C07304=1180.329,132.790,-53.848,-178.564,6.325,148.723
C07305=1180.334,132.522,-53.826,-178.567,6.323,148.724
C07306=1180.340,132.253,-53.804,-178.570,6.322,148.724
C07307=1180.345,131.985,-53.783,-178.573,6.320,148.725
C07308=1180.349,131.735,-53.763,-178.576,6.319,148.725
C07309=1180.354,131.487,-53.743,-178.578,6.318,148.726
C07310=1180.360,131.238,-53.722,-178.581,6.316,148.726
C07311=1180.364,130.988,-53.703,-178.583,6.314,148.726
C07312=1180.369,130.739,-53.682,-178.586,6.313,148.727
C07313=1180.374,130.489,-53.663,-178.589,6.311,148.727
C07314=1180.379,130.241,-53.643,-178.591,6.310,148.728
C07315=1180.383,129.992,-53.623,-178.594,6.308,148.728
C07316=1180.388,129.742,-53.603,-178.597,6.307,148.729
C07317=1180.392,129.493,-53.583,-178.600,6.305,148.729
C07318=1180.398,129.244,-53.564,-178.602,6.304,148.730
C07319=1180.402,128.995,-53.543,-178.605,6.302,148.730
C07320=1180.407,128.746,-53.524,-178.607,6.301,148.730
C07321=1180.411,128.497,-53.503,-178.611,6.299,148.731
C07322=1180.416,128.247,-53.484,-178.613,6.298,148.731
C07323=1180.422,127.998,-53.464,-178.615,6.297,148.732
C07324=1180.426,127.749,-53.444,-178.618,6.295,148.732
C07325=1180.431,127.500,-53.424,-178.621,6.294,148.733
C07326=1180.435,127.250,-53.405,-178.623,6.293,148.733
C07327=1180.440,127.002,-53.385,-178.626,6.291,148.734
C07328=1180.445,126.752,-53.365,-178.629,6.289,148.734
C07329=1180.450,126.503,-53.345,-178.631,6.289,148.735
C07330=1180.454,126.254,-53.325,-178.634,6.287,148.735
C07331=1180.460,126.005,-53.306,-178.637,6.285,148.735
C07332=1180.465,125.756,-53.286,-178.640,6.283,148.736
C07333=1180.469,125.507,-53.266,-178.642,6.283,148.736
C07334=1180.474,125.258,-53.246,-178.645,6.281,148.737
C07335=1180.479,125.008,-53.227,-178.648,6.279,148.737
C07336=1180.484,124.759,-53.207,-178.650,6.278,148.738
C07337=1180.488,124.510,-53.187,-178.653,6.277,148.738
C07338=1180.493,124.261,-53.168,-178.656,6.275,148.739
C07339=1180.498,124.012,-53.148,-178.658,6.273,148.739
C07340=1180.502,123.762,-53.129,-178.660,6.273,148.739
C07341=1180.508,123.513,-53.109,-178.664,6.271,148.740
C07342=1180.512,123.264,-53.089,-178.666,6.269,148.740
C07343=1180.517,123.015,-53.069,-178.669,6.268,148.741
C07344=1180.522,122.766,-53.050,-178.671,6.267,148.741
C07345=1180.527,122.516,-53.030,-178.674,6.265,148.742
C07346=1180.531,122.267,-53.011,-178.677,6.264,148.742
C07347=1180.536,122.018,-52.992,-178.679,6.263,148.743
C07348=1180.541,121.768,-52.972,-178.682,6.261,148.743
C07349=1180.545,121.519,-52.952,-178.685,6.260,148.744
C07350=1180.551,121.271,-52.933,-178.687,6.259,148.744
C07351=1180.556,121.021,-52.913,-178.690,6.257,148.745
C07352=1180.560,120.773,-52.894,-178.693,6.256,148.745
C07353=1180.565,120.523,-52.875,-178.695,6.255,148.746
C07354=1180.570,120.273,-52.855,-178.698,6.253,148.746
C07355=1180.575,120.024,-52.836,-178.701,6.251,148.747
C07356=1180.580,119.775,-52.816,-178.704,6.250,148.747
C07357=1180.584,119.526,-52.797,-178.706,6.249,148.747
C07358=1180.589,119.277,-52.778,-178.709,6.247,148.748
C07359=1180.594,119.027,-52.758,-178.712,6.246,148.748
C07360=1180.599,118.778,-52.739,-178.714,6.245,148.749
C07361=1180.603,118.529,-52.720,-178.717,6.243,148.749
C07362=1180.608,118.280,-52.700,-178.720,6.242,148.750
C07363=1180.613,118.031,-52.681,-178.722,6.241,148.750
C07364=1180.617,117.781,-52.662,-178.725,6.239,148.751
C07365=1180.623,117.533,-52.642,-178.727,6.237,148.751
C07366=1180.627,117.283,-52.623,-178.730,6.237,148.752
C07367=1180.633,117.034,-52.604,-178.733,6.235,148.752
C07368=1180.637,116.785,-52.584,-178.735,6.233,148.753
C07369=1180.642,116.536,-52.565,-178.738,6.233,148.753
C07370=1180.647,116.286,-52.546,-178.741,6.231,148.754
C07371=1180.652,116.037,-52.528,-178.743,6.229,148.754
C07372=1180.656,115.788,-52.508,-178.746,6.229,148.755
C07373=1180.661,115.538,-52.488,-178.749,6.227,148.755
C07374=1180.666,115.290,-52.470,-178.751,6.225,148.755
C07375=1180.671,115.040,-52.450,-178.753,6.224,148.756
C07376=1180.676,114.791,-52.431,-178.757,6.223,148.756
C07377=1180.680,114.542,-52.412,-178.759,6.221,148.757
C07378=1180.686,114.292,-52.393,-178.762,6.220,148.757
C07379=1180.690,114.043,-52.373,-178.765,6.219,148.758
C07380=1180.695,113.794,-52.355,-178.767,6.217,148.758
C07381=1180.700,113.545,-52.335,-178.770,6.216,148.759
C07382=1180.704,113.296,-52.316,-178.773,6.215,148.759
C07383=1180.709,113.046,-52.297,-178.775,6.214,148.760
C07384=1180.715,112.797,-52.278,-178.778,6.212,148.760
C07385=1180.719,112.549,-52.259,-178.781,6.211,148.761
C07386=1180.724,112.299,-52.240,-178.783,6.210,148.761
C07387=1180.729,112.050,-52.222,-178.786,6.208,148.762
C07388=1180.734,111.800,-52.202,-178.789,6.207,148.762
C07389=1180.738,111.552,-52.183,-178.791,6.206,148.763
C07390=1180.743,111.301,-52.164,-178.794,6.204,148.763
C07391=1180.748,111.053,-52.146,-178.797,6.203,148.764
C07392=1180.753,110.803,-52.126,-178.799,6.202,148.764
C07393=1180.758,110.554,-52.107,-178.802,6.200,148.764
C07394=1180.762,110.305,-52.088,-178.804,6.199,148.765
C07395=1180.768,110.056,-52.069,-178.807,6.198,148.766
C07396=1180.773,109.807,-52.051,-178.810,6.196,148.766
C07397=1180.777,109.557,-52.031,-178.812,6.195,148.767
C07398=1180.782,109.308,-52.013,-178.815,6.194,148.767
C07399=1180.786,109.059,-51.994,-178.817,6.193,148.767
C07400=1180.792,108.810,-51.975,-178.820,6.191,148.768
C07401=1180.796,108.560,-51.957,-178.823,6.190,148.768
C07402=1180.801,108.311,-51.938,-178.825,6.189,148.769
C07403=1180.806,108.062,-51.920,-178.828,6.187,148.769
C07404=1180.811,107.812,-51.900,-178.831,6.186,148.770
C07405=1180.815,107.564,-51.881,-178.834,6.185,148.771
C07406=1180.820,107.313,-51.862,-178.836,6.183,148.771
C07407=1180.825,107.065,-51.844,-178.839,6.182,148.771
C07408=1180.831,106.796,-51.824,-178.842,6.181,148.772
C07409=1180.835,106.527,-51.804,-178.844,6.179,148.772
C07410=1180.841,106.259,-51.783,-178.848,6.178,148.773
C07411=1180.846,105.991,-51.764,-178.850,6.176,148.773
C07412=1180.851,105.742,-51.744,-178.853,6.176,148.774
C07413=1180.856,105.492,-51.726,-178.856,6.174,148.774
C07414=1180.860,105.244,-51.707,-178.858,6.173,148.775
C07415=1180.865,104.994,-51.688,-178.861,6.172,148.776
C07416=1180.870,104.744,-51.670,-178.864,6.170,148.776
C07417=1180.876,104.496,-51.651,-178.866,6.169,148.777
C07418=1180.880,104.246,-51.633,-178.869,6.168,148.777
C07419=1180.884,103.997,-51.614,-178.871,6.167,148.777
C07420=1180.890,103.748,-51.595,-178.874,6.165,148.778
C07421=1180.895,103.499,-51.577,-178.876,6.164,148.778
C07422=1180.899,103.249,-51.558,-178.879,6.163,148.779
C07423=1180.905,103.000,-51.540,-178.882,6.161,148.779
C07424=1180.909,102.751,-51.521,-178.885,6.160,148.780
C07425=1180.914,102.501,-51.503,-178.888,6.159,148.781
C07426=1180.919,102.252,-51.485,-178.890,6.158,148.781
C07427=1180.924,102.003,-51.466,-178.893,6.156,148.781
C07428=1180.928,101.753,-51.447,-178.895,6.156,148.782
C07429=1180.933,101.504,-51.429,-178.898,6.154,148.782
C07430=1180.939,101.255,-51.411,-178.901,6.153,148.783
C07431=1180.943,101.006,-51.392,-178.903,6.152,148.783
C07432=1180.948,100.756,-51.374,-178.906,6.150,148.784
C07433=1180.953,100.507,-51.356,-178.909,6.150,148.785
C07434=1180.958,100.258,-51.336,-178.911,6.148,148.785
C07435=1180.963,100.009,-51.318,-178.914,6.147,148.786
C07436=1180.967,99.759,-51.300,-178.917,6.146,148.786
C07437=1180.972,99.510,-51.282,-178.919,6.145,148.786
C07438=1180.977,99.261,-51.264,-178.922,6.143,148.787
C07439=1180.982,99.012,-51.245,-178.925,6.142,148.787
C07440=1180.987,98.762,-51.226,-178.927,6.141,148.788
C07441=1180.992,98.513,-51.208,-178.930,6.139,148.789
C07442=1180.996,98.264,-51.190,-178.932,6.138,148.789
C07443=1181.001,98.015,-51.172,-178.935,6.137,148.790
C07444=1181.006,97.765,-51.153,-178.937,6.136,148.790
C07445=1181.011,97.516,-51.135,-178.941,6.135,148.791
C07446=1181.016,97.267,-51.117,-178.943,6.134,148.791
C07447=1181.021,97.018,-51.099,-178.946,6.132,148.791
C07448=1181.026,96.768,-51.081,-178.948,6.132,148.792
C07449=1181.030,96.518,-51.063,-178.951,6.130,148.793
C07450=1181.035,96.269,-51.045,-178.953,6.129,148.793
C07451=1181.041,96.020,-51.026,-178.956,6.128,148.794
C07452=1181.046,95.771,-51.008,-178.959,6.126,148.794
C07453=1181.050,95.521,-50.990,-178.962,6.125,148.795
C07454=1181.055,95.273,-50.971,-178.964,6.124,148.795
C07455=1181.059,95.023,-50.953,-178.967,6.123,148.796
C07456=1181.064,94.774,-50.935,-178.970,6.121,148.796
C07457=1181.069,94.525,-50.917,-178.972,6.120,148.797
C07458=1181.074,94.276,-50.899,-178.975,6.119,148.797
C07459=1181.079,94.026,-50.881,-178.977,6.118,148.798
C07460=1181.084,93.777,-50.863,-178.980,6.117,148.798
C07461=1181.088,93.527,-50.845,-178.982,6.116,148.799
C07462=1181.093,93.278,-50.827,-178.986,6.114,148.799
C07463=1181.098,93.029,-50.809,-178.988,6.114,148.800
C07464=1181.103,92.780,-50.791,-178.990,6.112,148.800
C07465=1181.109,92.530,-50.773,-178.993,6.111,148.801
C07466=1181.114,92.280,-50.755,-178.996,6.110,148.801
C07467=1181.119,92.031,-50.737,-178.998,6.109,148.802
C07468=1181.124,91.782,-50.719,-179.001,6.107,148.802
C07469=1181.128,91.532,-50.701,-179.004,6.107,148.803
C07470=1181.133,91.283,-50.683,-179.006,6.105,148.803
C07471=1181.138,91.034,-50.665,-179.009,6.104,148.804
C07472=1181.142,90.785,-50.647,-179.012,6.103,148.804
C07473=1181.147,90.536,-50.629,-179.014,6.102,148.805
C07474=1181.152,90.287,-50.611,-179.017,6.100,148.805
C07475=1181.157,90.037,-50.594,-179.019,6.100,148.806
C07476=1181.162,89.788,-50.576,-179.022,6.098,148.807
C07477=1181.167,89.539,-50.558,-179.025,6.097,148.807
C07478=1181.172,89.289,-50.540,-179.028,6.096,148.808
C07479=1181.177,89.040,-50.522,-179.030,6.095,148.808
C07480=1181.182,88.791,-50.504,-179.033,6.094,148.809
C07481=1181.187,88.541,-50.487,-179.035,6.093,148.809
C07482=1181.191,88.291,-50.469,-179.038,6.091,148.810
C07483=1181.196,88.042,-50.451,-179.041,6.091,148.810
C07484=1181.201,87.793,-50.433,-179.043,6.089,148.811
C07485=1181.206,87.543,-50.415,-179.046,6.088,148.811
C07486=1181.211,87.294,-50.397,-179.049,6.087,148.812
C07487=1181.215,87.045,-50.380,-179.051,6.086,148.812
C07488=1181.220,86.796,-50.362,-179.054,6.084,148.813
C07489=1181.225,86.546,-50.345,-179.057,6.084,148.813
C07490=1181.230,86.297,-50.327,-179.059,6.083,148.814
C07491=1181.235,86.048,-50.309,-179.062,6.082,148.814
C07492=1181.240,85.798,-50.292,-179.064,6.081,148.815
C07493=1181.245,85.549,-50.274,-179.067,6.079,148.815
C07494=1181.249,85.300,-50.256,-179.069,6.078,148.816
C07495=1181.255,85.050,-50.239,-179.072,6.077,148.816
C07496=1181.260,84.801,-50.221,-179.075,6.076,148.817
C07497=1181.265,84.552,-50.203,-179.078,6.074,148.817
C07498=1181.270,84.302,-50.186,-179.080,6.074,148.818
C07499=1181.274,84.053,-50.168,-179.083,6.072,148.819
C07500=1181.279,83.804,-50.150,-179.086,6.072,148.819
C07501=1181.284,83.554,-50.133,-179.088,6.071,148.820
C07502=1181.289,83.305,-50.115,-179.091,6.069,148.820
C07503=1181.294,83.055,-50.098,-179.093,6.068,148.821
C07504=1181.298,82.806,-50.080,-179.096,6.067,148.821
C07505=1181.304,82.557,-50.063,-179.098,6.066,148.822
C07506=1181.309,82.308,-50.046,-179.102,6.065,148.822
C07507=1181.314,82.059,-50.028,-179.104,6.064,148.823
C07508=1181.318,81.809,-50.011,-179.107,6.063,148.823
C07509=1181.323,81.560,-49.993,-179.109,6.062,148.824
C07510=1181.329,81.310,-49.976,-179.111,6.061,148.824
C07511=1181.333,81.062,-49.958,-179.114,6.059,148.825
C07512=1181.338,80.793,-49.940,-179.118,6.058,148.826
C07513=1181.344,80.524,-49.921,-179.120,6.057,148.826
C07514=1181.349,80.256,-49.902,-179.123,6.056,148.827
C07515=1181.355,79.987,-49.883,-179.126,6.055,148.827
C07516=1181.359,79.739,-49.866,-179.128,6.054,148.828
C07517=1181.364,79.489,-49.848,-179.131,6.053,148.828
C07518=1181.369,79.239,-49.831,-179.134,6.051,148.829
C07519=1181.373,78.990,-49.814,-179.136,6.051,148.830
C07520=1181.379,78.741,-49.797,-179.138,6.050,148.830
C07521=1181.384,78.492,-49.779,-179.142,6.049,148.831
C07522=1181.389,78.242,-49.762,-179.144,6.048,148.831
C07523=1181.394,77.993,-49.745,-179.147,6.046,148.832
C07524=1181.399,77.743,-49.727,-179.149,6.045,148.832
C07525=1181.403,77.494,-49.710,-179.152,6.044,148.833
C07526=1181.408,77.245,-49.692,-179.154,6.043,148.833
C07527=1181.413,76.995,-49.676,-179.157,6.043,148.834
C07528=1181.418,76.746,-49.659,-179.160,6.041,148.834
C07529=1181.423,76.497,-49.641,-179.162,6.040,148.835
C07530=1181.428,76.248,-49.624,-179.165,6.039,148.835
C07531=1181.433,75.998,-49.607,-179.168,6.038,148.836
C07532=1181.438,75.748,-49.590,-179.170,6.037,148.836
C07533=1181.442,75.499,-49.572,-179.173,6.036,148.837
C07534=1181.448,75.250,-49.556,-179.175,6.035,148.838
C07535=1181.453,75.000,-49.539,-179.179,6.034,148.838
C07536=1181.458,74.751,-49.521,-179.181,6.033,148.839
C07537=1181.462,74.502,-49.504,-179.183,6.032,148.839
C07538=1181.467,74.252,-49.487,-179.186,6.031,148.840
C07539=1181.472,74.003,-49.470,-179.189,6.030,148.840
C07540=1181.477,73.754,-49.453,-179.191,6.028,148.841
C07541=1181.482,73.505,-49.436,-179.194,6.028,148.841
C07542=1181.487,73.255,-49.419,-179.196,6.027,148.842
C07543=1181.492,73.005,-49.402,-179.199,6.025,148.843
C07544=1181.497,72.756,-49.385,-179.201,6.025,148.843
C07545=1181.502,72.507,-49.368,-179.204,6.024,148.844
C07546=1181.507,72.258,-49.350,-179.207,6.022,148.844
C07547=1181.511,72.008,-49.334,-179.209,6.022,148.845
C07548=1181.516,71.758,-49.316,-179.212,6.020,148.845
C07549=1181.522,71.509,-49.300,-179.215,6.020,148.846
C07550=1181.527,71.260,-49.283,-179.217,6.019,148.846
C07551=1181.531,71.010,-49.266,-179.220,6.017,148.847
C07552=1181.536,70.761,-49.248,-179.222,6.016,148.847
C07553=1181.541,70.512,-49.232,-179.225,6.016,148.848
C07554=1181.546,70.263,-49.215,-179.228,6.015,148.849
C07555=1181.551,70.013,-49.198,-179.230,6.014,148.849
C07556=1181.555,69.763,-49.181,-179.234,6.012,148.850
C07557=1181.561,69.514,-49.164,-179.236,6.011,148.850
C07558=1181.566,69.265,-49.148,-179.238,6.011,148.851
C07559=1181.571,69.015,-49.130,-179.241,6.009,148.851
C07560=1181.576,68.766,-49.114,-179.244,6.009,148.852
C07561=1181.580,68.517,-49.097,-179.246,6.008,148.852
C07562=1181.586,68.267,-49.080,-179.249,6.006,148.853
C07563=1181.590,68.018,-49.064,-179.251,6.006,148.853
C07564=1181.595,67.769,-49.047,-179.254,6.005,148.854
C07565=1181.600,67.519,-49.030,-179.257,6.003,148.855
C07566=1181.605,67.269,-49.013,-179.259,6.003,148.855
C07567=1181.610,67.021,-48.997,-179.262,6.002,148.856
C07568=1181.615,66.771,-48.980,-179.265,6.001,148.856
C07569=1181.620,66.521,-48.963,-179.267,6.000,148.857
C07570=1181.625,66.273,-48.947,-179.270,5.998,148.857
C07571=1181.630,66.023,-48.930,-179.273,5.998,148.858
C07572=1181.634,65.773,-48.913,-179.275,5.997,148.858
C07573=1181.640,65.525,-48.897,-179.278,5.996,148.859
C07574=1181.645,65.275,-48.879,-179.280,5.995,148.860
C07575=1181.649,65.025,-48.863,-179.283,5.994,148.860
C07576=1181.655,64.776,-48.847,-179.285,5.993,148.861
C07577=1181.660,64.526,-48.830,-179.288,5.992,148.861
C07578=1181.664,64.277,-48.813,-179.291,5.991,148.862
C07579=1181.669,64.028,-48.797,-179.293,5.990,148.862
C07580=1181.674,63.778,-48.780,-179.296,5.989,148.863
C07581=1181.679,63.529,-48.763,-179.298,5.988,148.863
C07582=1181.684,63.280,-48.747,-179.301,5.987,148.864
C07583=1181.689,63.030,-48.731,-179.304,5.986,148.865
C07584=1181.694,62.781,-48.714,-179.306,5.986,148.865
C07585=1181.699,62.531,-48.697,-179.308,5.985,148.866
C07586=1181.704,62.282,-48.680,-179.312,5.983,148.866
C07587=1181.709,62.033,-48.664,-179.314,5.983,148.867
C07588=1181.714,61.783,-48.648,-179.316,5.982,148.867
C07589=1181.719,61.534,-48.632,-179.320,5.981,148.868
C07590=1181.724,61.284,-48.615,-179.322,5.980,148.869
C07591=1181.728,61.035,-48.598,-179.324,5.979,148.869
C07592=1181.734,60.785,-48.582,-179.327,5.978,148.870
C07593=1181.738,60.536,-48.566,-179.330,5.977,148.870
C07594=1181.743,60.287,-48.549,-179.332,5.976,148.871
C07595=1181.749,60.037,-48.532,-179.335,5.975,148.871
C07596=1181.754,59.788,-48.516,-179.338,5.974,148.872
C07597=1181.758,59.538,-48.500,-179.340,5.973,148.872
C07598=1181.763,59.289,-48.483,-179.343,5.972,148.873
C07599=1181.768,59.039,-48.468,-179.345,5.971,148.874
C07600=1181.773,58.790,-48.451,-179.348,5.971,148.874
C07601=1181.779,58.541,-48.434,-179.350,5.970,148.875
C07602=1181.783,58.291,-48.418,-179.353,5.968,148.875
C07603=1181.788,58.042,-48.402,-179.356,5.968,148.876
C07604=1181.793,57.792,-48.385,-179.358,5.967,148.876
C07605=1181.798,57.543,-48.369,-179.361,5.966,148.877
C07606=1181.803,57.294,-48.353,-179.363,5.965,148.878
C07607=1181.808,57.044,-48.337,-179.366,5.964,148.878
C07608=1181.813,56.795,-48.321,-179.369,5.964,148.879
C07609=1181.818,56.546,-48.304,-179.371,5.962,148.879
C07610=1181.823,56.296,-48.288,-179.374,5.962,148.880
C07611=1181.828,56.047,-48.271,-179.376,5.961,148.880
C07612=1181.833,55.797,-48.255,-179.379,5.959,148.881
C07613=1181.838,55.548,-48.239,-179.381,5.958,148.882
C07614=1181.843,55.298,-48.223,-179.384,5.958,148.882
C07615=1181.848,55.049,-48.207,-179.387,5.957,148.883
C07616=1181.853,54.780,-48.189,-179.389,5.956,148.883
C07617=1181.859,54.511,-48.172,-179.392,5.955,148.884
C07618=1181.864,54.243,-48.155,-179.395,5.954,148.885
C07619=1181.869,53.975,-48.138,-179.398,5.953,148.885
C07620=1181.874,53.725,-48.122,-179.400,5.952,148.886
C07621=1181.879,53.476,-48.105,-179.403,5.951,148.886
C07622=1181.884,53.226,-48.089,-179.406,5.951,148.887
C07623=1181.889,52.977,-48.073,-179.408,5.950,148.888
C07624=1181.894,52.727,-48.057,-179.411,5.949,148.888
C07625=1181.899,52.478,-48.041,-179.414,5.948,148.889
C07626=1181.904,52.228,-48.025,-179.416,5.947,148.889
C07627=1181.909,51.979,-48.009,-179.419,5.947,148.890
C07628=1181.914,51.730,-47.993,-179.422,5.945,148.890
C07629=1181.919,51.480,-47.977,-179.424,5.944,148.891
C07630=1181.924,51.231,-47.961,-179.426,5.943,148.892
C07631=1181.929,50.981,-47.945,-179.429,5.943,148.892
C07632=1181.934,50.732,-47.929,-179.432,5.941,148.893
C07633=1181.939,50.482,-47.913,-179.434,5.941,148.893
C07634=1181.944,50.233,-47.897,-179.437,5.940,148.894
C07635=1181.949,49.984,-47.881,-179.439,5.939,148.894
C07636=1181.953,49.734,-47.865,-179.442,5.938,148.895
C07637=1181.959,49.485,-47.850,-179.445,5.938,148.896
C07638=1181.963,49.235,-47.833,-179.447,5.937,148.896
C07639=1181.969,48.986,-47.818,-179.450,5.936,148.897
C07640=1181.974,48.736,-47.802,-179.452,5.935,148.897
C07641=1181.978,48.487,-47.785,-179.455,5.934,148.898
C07642=1181.984,48.238,-47.770,-179.458,5.933,148.899
C07643=1181.989,47.988,-47.754,-179.460,5.933,148.899
C07644=1181.993,47.738,-47.739,-179.463,5.932,148.900
C07645=1181.998,47.490,-47.722,-179.465,5.930,148.900
C07646=1182.003,47.239,-47.706,-179.468,5.930,148.901
C07647=1182.009,46.990,-47.691,-179.471,5.929,148.902
C07648=1182.014,46.741,-47.675,-179.473,5.928,148.902
C07649=1182.018,46.491,-47.659,-179.476,5.927,148.903
C07650=1182.023,46.242,-47.644,-179.478,5.926,148.903
C07651=1182.028,45.993,-47.628,-179.481,5.926,148.904
C07652=1182.033,45.743,-47.612,-179.483,5.925,148.904
C07653=1182.039,45.493,-47.597,-179.486,5.924,148.905
C07654=1182.044,45.244,-47.580,-179.489,5.923,148.906
C07655=1182.048,44.995,-47.565,-179.491,5.922,148.906
C07656=1182.053,44.745,-47.549,-179.494,5.922,148.907
C07657=1182.059,44.496,-47.534,-179.496,5.921,148.907
C07658=1182.064,44.246,-47.518,-179.499,5.919,148.908
C07659=1182.068,43.997,-47.503,-179.502,5.919,148.908
C07660=1182.073,43.747,-47.487,-179.504,5.918,148.909
C07661=1182.079,43.498,-47.472,-179.506,5.918,148.910
C07662=1182.083,43.248,-47.455,-179.509,5.917,148.910
C07663=1182.088,42.999,-47.440,-179.512,5.915,148.911
C07664=1182.093,42.750,-47.424,-179.514,5.915,148.911
C07665=1182.099,42.500,-47.409,-179.517,5.914,148.912
C07666=1182.103,42.250,-47.393,-179.519,5.913,148.912
C07667=1182.108,42.001,-47.378,-179.522,5.913,148.913
C07668=1182.113,41.752,-47.362,-179.525,5.912,148.914
C07669=1182.118,41.502,-47.346,-179.527,5.911,148.914
C07670=1182.123,41.253,-47.331,-179.530,5.910,148.915
C07671=1182.128,41.003,-47.316,-179.532,5.909,148.915
C07672=1182.134,40.754,-47.300,-179.535,5.909,148.916
C07673=1182.138,40.504,-47.284,-179.538,5.908,148.917
C07674=1182.143,40.255,-47.269,-179.540,5.907,148.917
C07675=1182.148,40.005,-47.254,-179.543,5.906,148.918
C07676=1182.154,39.756,-47.238,-179.545,5.906,148.918
C07677=1182.159,39.507,-47.223,-179.547,5.905,148.919
C07678=1182.163,39.257,-47.207,-179.550,5.904,148.920
C07679=1182.169,39.007,-47.191,-179.553,5.903,148.920
C07680=1182.173,38.758,-47.176,-179.556,5.902,148.921
C07681=1182.179,38.509,-47.161,-179.558,5.902,148.921
C07682=1182.183,38.259,-47.145,-179.560,5.901,148.922
C07683=1182.188,38.010,-47.130,-179.563,5.900,148.923
C07684=1182.194,37.760,-47.114,-179.566,5.900,148.923
C07685=1182.198,37.511,-47.099,-179.568,5.898,148.924
C07686=1182.204,37.261,-47.084,-179.571,5.898,148.924
C07687=1182.209,37.012,-47.069,-179.574,5.897,148.925
C07688=1182.213,36.762,-47.053,-179.576,5.896,148.925
C07689=1182.219,36.512,-47.038,-179.578,5.896,148.926
C07690=1182.223,36.263,-47.023,-179.582,5.894,148.927
C07691=1182.229,36.014,-47.007,-179.584,5.893,148.927
C07692=1182.233,35.765,-46.992,-179.586,5.893,148.928
C07693=1182.239,35.515,-46.977,-179.589,5.892,148.928
C07694=1182.243,35.265,-46.962,-179.591,5.892,148.929
C07695=1182.249,35.016,-46.946,-179.594,5.891,148.930
C07696=1182.254,34.766,-46.931,-179.596,5.890,148.930
C07697=1182.259,34.517,-46.916,-179.599,5.889,148.931
C07698=1182.264,34.267,-46.901,-179.602,5.888,148.931
C07699=1182.269,34.018,-46.886,-179.604,5.888,148.932
C07700=1182.274,33.768,-46.870,-179.607,5.887,148.933
C07701=1182.278,33.519,-46.855,-179.609,5.887,148.933
C07702=1182.284,33.269,-46.840,-179.612,5.886,148.934
C07703=1182.289,33.020,-46.825,-179.615,5.884,148.934
C07704=1182.294,32.770,-46.810,-179.617,5.884,148.935
C07705=1182.299,32.521,-46.795,-179.620,5.883,148.936
C07706=1182.304,32.271,-46.780,-179.622,5.883,148.936
C07707=1182.309,32.022,-46.765,-179.625,5.882,148.937
C07708=1182.314,31.773,-46.749,-179.627,5.881,148.937
C07709=1182.319,31.522,-46.735,-179.630,5.881,148.938
C07710=1182.323,31.273,-46.720,-179.633,5.879,148.939
C07711=1182.329,31.024,-46.704,-179.635,5.878,148.939
C07712=1182.334,30.774,-46.690,-179.638,5.878,148.940
C07713=1182.339,30.525,-46.674,-179.640,5.877,148.940
C07714=1182.344,30.276,-46.659,-179.642,5.877,148.941
C07715=1182.350,30.026,-46.644,-179.645,5.876,148.942
C07716=1182.354,29.776,-46.629,-179.647,5.875,148.942
C07717=1182.359,29.527,-46.614,-179.650,5.875,148.943
C07718=1182.365,29.277,-46.599,-179.653,5.873,148.943
C07719=1182.369,29.028,-46.584,-179.655,5.873,148.944
C07720=1182.375,28.759,-46.568,-179.658,5.872,148.945
C07721=1182.380,28.490,-46.552,-179.661,5.872,148.945
C07722=1182.386,28.221,-46.536,-179.664,5.870,148.946
C07723=1182.391,27.953,-46.520,-179.666,5.870,148.947
C07724=1182.396,27.703,-46.505,-179.669,5.869,148.947
C07725=1182.401,27.454,-46.490,-179.671,5.868,148.948
C07726=1182.406,27.204,-46.476,-179.674,5.868,148.948
C07727=1182.411,26.955,-46.461,-179.677,5.867,148.949
C07728=1182.416,26.705,-46.446,-179.679,5.867,148.950
C07729=1182.421,26.456,-46.431,-179.682,5.865,148.950
C07730=1182.426,26.206,-46.416,-179.685,5.865,148.951
C07731=1182.431,25.957,-46.401,-179.687,5.864,148.951
C07732=1182.436,25.707,-46.387,-179.689,5.863,148.952
C07733=1182.441,25.458,-46.372,-179.692,5.863,148.953
C07734=1182.447,25.208,-46.357,-179.694,5.862,148.953
C07735=1182.451,24.959,-46.342,-179.697,5.862,148.954
C07736=1182.456,24.709,-46.327,-179.700,5.861,148.955
C07737=1182.462,24.460,-46.312,-179.702,5.860,148.955
C07738=1182.467,24.210,-46.298,-179.704,5.860,148.956
C07739=1182.472,23.961,-46.283,-179.708,5.858,148.956
C07740=1182.476,23.711,-46.268,-179.710,5.858,148.957
C07741=1182.482,23.461,-46.253,-179.712,5.857,148.957
C07742=1182.487,23.212,-46.238,-179.715,5.857,148.958
C07743=1182.492,22.963,-46.224,-179.717,5.856,148.959
C07744=1182.497,22.713,-46.210,-179.720,5.855,148.959
C07745=1182.502,22.464,-46.194,-179.722,5.855,148.960
C07746=1182.507,22.214,-46.180,-179.725,5.854,148.960
C07747=1182.512,21.965,-46.165,-179.727,5.853,148.961
C07748=1182.516,21.715,-46.151,-179.730,5.853,148.962
C07749=1182.521,21.465,-46.136,-179.732,5.852,148.962
C07750=1182.527,21.216,-46.121,-179.735,5.851,148.963
C07751=1182.532,20.966,-46.107,-179.738,5.850,148.964
C07752=1182.537,20.716,-46.092,-179.740,5.849,148.964
C07753=1182.541,20.467,-46.077,-179.743,5.849,148.965
C07754=1182.546,20.218,-46.063,-179.745,5.848,148.965
C07755=1182.553,19.968,-46.049,-179.748,5.848,148.966
C07756=1182.558,19.719,-46.034,-179.750,5.847,148.967
C07757=1182.562,19.470,-46.019,-179.753,5.847,148.967
C07758=1182.567,19.220,-46.005,-179.755,5.846,148.968
C07759=1182.572,18.970,-45.991,-179.758,5.845,148.968
C07760=1182.577,18.720,-45.976,-179.760,5.845,148.969
C07761=1182.582,18.471,-45.961,-179.763,5.844,148.969
C07762=1182.587,18.221,-45.947,-179.765,5.843,148.970
C07763=1182.592,17.972,-45.932,-179.768,5.843,148.971
C07764=1182.598,17.723,-45.918,-179.771,5.842,148.972
C07765=1182.603,17.473,-45.903,-179.773,5.841,148.972
C07766=1182.608,17.224,-45.889,-179.776,5.840,148.973
C07767=1182.613,16.974,-45.875,-179.779,5.840,148.973
C07768=1182.617,16.724,-45.861,-179.781,5.839,148.974
C07769=1182.622,16.475,-45.846,-179.783,5.838,148.974
C07770=1182.628,16.225,-45.831,-179.786,5.838,148.975
C07771=1182.633,15.976,-45.816,-179.788,5.837,148.976
C07772=1182.638,15.727,-45.802,-179.791,5.837,148.976
C07773=1182.643,15.477,-45.788,-179.793,5.836,148.977
C07774=1182.648,15.227,-45.774,-179.796,5.835,148.977
C07775=1182.653,14.977,-45.760,-179.798,5.835,148.978
C07776=1182.658,14.728,-45.745,-179.801,5.834,148.979
C07777=1182.663,14.478,-45.731,-179.803,5.833,148.979
C07778=1182.669,14.229,-45.717,-179.806,5.833,148.980
C07779=1182.673,13.980,-45.702,-179.808,5.832,148.981
C07780=1182.678,13.730,-45.688,-179.811,5.832,148.981
C07781=1182.683,13.480,-45.674,-179.813,5.831,148.982
C07782=1182.688,13.231,-45.659,-179.816,5.831,148.982
C07783=1182.694,12.982,-45.645,-179.818,5.830,148.983
C07784=1182.699,12.732,-45.631,-179.821,5.829,148.984
C07785=1182.704,12.482,-45.617,-179.824,5.828,148.984
C07786=1182.709,12.233,-45.603,-179.827,5.828,148.985
C07787=1182.714,11.983,-45.588,-179.829,5.827,148.985
C07788=1182.719,11.734,-45.574,-179.831,5.826,148.986
C07789=1182.724,11.484,-45.560,-179.834,5.826,148.987
C07790=1182.729,11.234,-45.546,-179.836,5.825,148.987
C07791=1182.734,10.985,-45.532,-179.839,5.824,148.988
C07792=1182.740,10.736,-45.518,-179.841,5.824,148.989
C07793=1182.744,10.486,-45.503,-179.844,5.823,148.989
C07794=1182.749,10.236,-45.489,-179.846,5.823,148.990
C07795=1182.754,9.987,-45.475,-179.849,5.822,148.990
C07796=1182.760,9.738,-45.461,-179.852,5.822,148.991
C07797=1182.765,9.488,-45.447,-179.854,5.821,148.992
C07798=1182.770,9.238,-45.432,-179.856,5.820,148.992
C07799=1182.775,8.988,-45.418,-179.859,5.820,148.993
C07800=1182.780,8.739,-45.405,-179.861,5.819,148.993
C07801=1182.785,8.489,-45.391,-179.864,5.818,148.994
C07802=1182.790,8.240,-45.377,-179.867,5.818,148.995
C07803=1182.795,7.990,-45.363,-179.869,5.817,148.995
C07804=1182.800,7.741,-45.349,-179.871,5.817,148.996
C07805=1182.805,7.491,-45.334,-179.874,5.816,148.997
C07806=1182.810,7.242,-45.320,-179.877,5.816,148.997
C07807=1182.815,6.992,-45.306,-179.879,5.815,148.998
C07808=1182.820,6.743,-45.293,-179.881,5.814,148.998
C07809=1182.825,6.493,-45.279,-179.884,5.814,148.999
C07810=1182.830,6.243,-45.265,-179.886,5.813,149.000
C07811=1182.836,5.994,-45.251,-179.889,5.813,149.000
C07812=1182.841,5.744,-45.237,-179.892,5.812,149.001
C07813=1182.846,5.495,-45.222,-179.894,5.811,149.001
C07814=1182.852,5.245,-45.209,-179.896,5.811,149.002
C07815=1182.856,4.996,-45.195,-179.899,5.810,149.003
C07816=1182.861,4.746,-45.181,-179.902,5.810,149.003
C07817=1182.866,4.497,-45.167,-179.904,5.809,149.004
C07818=1182.872,4.247,-45.154,-179.907,5.808,149.005
C07819=1182.877,3.997,-45.139,-179.909,5.808,149.005
C07820=1182.881,3.748,-45.126,-179.911,5.807,149.006
C07821=1182.886,3.499,-45.112,-179.914,5.807,149.006
C07822=1182.892,3.248,-45.098,-179.917,5.806,149.007
C07823=1182.897,2.999,-45.084,-179.919,5.805,149.008
C07824=1182.903,2.730,-45.069,-179.921,5.805,149.008
C07825=1182.907,2.461,-45.055,-179.924,5.804,149.009
C07826=1182.913,2.191,-45.040,-179.927,5.804,149.010
C07827=1182.919,1.923,-45.025,-179.929,5.803,149.010
C07828=1182.924,1.673,-45.011,-179.932,5.803,149.011
C07829=1182.929,1.423,-44.997,-179.935,5.803,149.012
C07830=1182.934,1.173,-44.984,-179.937,5.802,149.012
C07831=1182.939,0.924,-44.970,-179.940,5.801,149.013
C07832=1182.944,0.674,-44.956,-179.942,5.801,149.014
C07833=1182.950,0.425,-44.942,-179.944,5.800,149.014
C07834=1182.954,0.175,-44.929,-179.947,5.799,149.015
C07835=1182.960,-0.074,-44.916,-179.950,5.799,149.015
C07836=1182.965,-0.324,-44.901,-179.952,5.798,149.016
C07837=1182.969,-0.573,-44.888,-179.955,5.798,149.017
C07838=1182.975,-0.823,-44.874,-179.957,5.797,149.017
C07839=1182.980,-1.073,-44.860,-179.960,5.797,149.018
C07840=1182.985,-1.322,-44.847,-179.962,5.796,149.018
C07841=1182.990,-1.572,-44.833,-179.965,5.795,149.019
C07842=1182.995,-1.821,-44.819,-179.967,5.795,149.020
C07843=1183.000,-2.071,-44.806,-179.969,5.794,149.020
C07844=1183.005,-2.321,-44.792,-179.972,5.794,149.021
C07845=1183.011,-2.570,-44.779,-179.975,5.793,149.022
C07846=1183.015,-2.820,-44.765,-179.977,5.793,149.022
C07847=1183.021,-3.069,-44.752,-179.980,5.792,149.023
C07848=1183.026,-3.319,-44.738,-179.982,5.791,149.023
C07849=1183.031,-3.568,-44.725,-179.985,5.791,149.024
C07850=1183.036,-3.818,-44.711,-179.987,5.790,149.025
C07851=1183.042,-4.068,-44.698,-179.990,5.790,149.025
C07852=1183.046,-4.317,-44.684,-179.992,5.789,149.026
C07853=1183.052,-4.567,-44.671,-179.994,5.789,149.027
C07854=1183.056,-4.816,-44.657,-179.997,5.789,149.027
C07855=1183.061,-5.066,-44.644,-179.999,5.788,149.028
C07856=1183.067,-5.315,-44.630,179.998,5.788,149.029
C07857=1183.071,-5.565,-44.617,179.996,5.787,149.029
C07858=1183.077,-5.815,-44.603,179.993,5.786,149.030
C07859=1183.081,-6.064,-44.590,179.991,5.786,149.030
C07860=1183.087,-6.314,-44.577,179.988,5.785,149.031
C07861=1183.091,-6.563,-44.563,179.986,5.785,149.032
C07862=1183.097,-6.813,-44.550,179.983,5.784,149.032
C07863=1183.101,-7.062,-44.536,179.980,5.784,149.033
C07864=1183.107,-7.312,-44.523,179.978,5.783,149.033
C07865=1183.113,-7.562,-44.509,179.976,5.782,149.034
C07866=1183.117,-7.811,-44.496,179.973,5.782,149.035
C07867=1183.123,-8.061,-44.482,179.970,5.781,149.035
C07868=1183.128,-8.311,-44.470,179.968,5.781,149.036
C07869=1183.133,-8.560,-44.456,179.966,5.781,149.037
C07870=1183.138,-8.810,-44.443,179.963,5.780,149.037
C07871=1183.144,-9.059,-44.430,179.961,5.780,149.038
C07872=1183.148,-9.309,-44.416,179.959,5.779,149.038
C07873=1183.154,-9.558,-44.403,179.956,5.779,149.039
C07874=1183.158,-9.808,-44.390,179.953,5.778,149.040
C07875=1183.163,-10.057,-44.377,179.951,5.777,149.040
C07876=1183.168,-10.307,-44.363,179.948,5.777,149.041
C07877=1183.173,-10.557,-44.350,179.946,5.776,149.042
C07878=1183.179,-10.807,-44.337,179.944,5.776,149.042
C07879=1183.184,-11.056,-44.324,179.941,5.775,149.043
C07880=1183.189,-11.305,-44.310,179.938,5.775,149.044
C07881=1183.194,-11.555,-44.297,179.936,5.775,149.044
C07882=1183.200,-11.805,-44.284,179.934,5.774,149.045
C07883=1183.204,-12.054,-44.270,179.931,5.774,149.045
C07884=1183.209,-12.304,-44.258,179.929,5.773,149.046
C07885=1183.214,-12.554,-44.244,179.927,5.772,149.047
C07886=1183.220,-12.803,-44.232,179.924,5.772,149.047
C07887=1183.225,-13.052,-44.218,179.921,5.771,149.048
C07888=1183.230,-13.302,-44.205,179.919,5.771,149.049
C07889=1183.235,-13.552,-44.192,179.916,5.770,149.049
C07890=1183.240,-13.802,-44.179,179.914,5.770,149.050
C07891=1183.245,-14.051,-44.166,179.911,5.769,149.050
C07892=1183.251,-14.301,-44.153,179.909,5.770,149.051
C07893=1183.255,-14.550,-44.139,179.907,5.769,149.052
C07894=1183.260,-14.800,-44.127,179.904,5.768,149.052
C07895=1183.266,-15.049,-44.113,179.902,5.768,149.053
C07896=1183.271,-15.299,-44.100,179.899,5.767,149.053
C07897=1183.276,-15.549,-44.088,179.897,5.767,149.054
C07898=1183.281,-15.799,-44.074,179.894,5.766,149.055
C07899=1183.286,-16.048,-44.062,179.891,5.766,149.056
C07900=1183.291,-16.298,-44.049,179.889,5.765,149.056
C07901=1183.296,-16.547,-44.035,179.887,5.765,149.057
C07902=1183.301,-16.797,-44.022,179.884,5.765,149.057
C07903=1183.307,-17.046,-44.010,179.882,5.764,149.058
C07904=1183.312,-17.296,-43.996,179.880,5.763,149.059
C07905=1183.317,-17.546,-43.983,179.877,5.763,149.059
C07906=1183.322,-17.795,-43.971,179.874,5.762,149.060
C07907=1183.327,-18.045,-43.957,179.872,5.762,149.060
C07908=1183.332,-18.295,-43.945,179.869,5.761,149.061
C07909=1183.338,-18.544,-43.932,179.867,5.761,149.062
C07910=1183.342,-18.794,-43.919,179.865,5.761,149.062
C07911=1183.348,-19.044,-43.906,179.863,5.760,149.063
C07912=1183.353,-19.293,-43.893,179.860,5.760,149.064
C07913=1183.358,-19.542,-43.881,179.857,5.759,149.064
C07914=1183.363,-19.793,-43.867,179.855,5.758,149.065
C07915=1183.369,-20.042,-43.855,179.852,5.758,149.066
C07916=1183.374,-20.291,-43.842,179.850,5.758,149.066
C07917=1183.378,-20.541,-43.829,179.848,5.757,149.067
C07918=1183.384,-20.791,-43.816,179.846,5.757,149.067
C07919=1183.389,-21.040,-43.803,179.843,5.757,149.068
C07920=1183.394,-21.289,-43.791,179.840,5.756,149.069
C07921=1183.399,-21.540,-43.778,179.838,5.755,149.069
C07922=1183.404,-21.789,-43.765,179.835,5.755,149.070
C07923=1183.410,-22.039,-43.753,179.833,5.754,149.071
C07924=1183.415,-22.289,-43.740,179.831,5.754,149.071
C07925=1183.420,-22.538,-43.727,179.828,5.754,149.072
C07926=1183.425,-22.788,-43.714,179.826,5.753,149.072
C07927=1183.430,-23.037,-43.702,179.823,5.753,149.073
C07928=1183.436,-23.307,-43.687,179.820,5.753,149.074
C07929=1183.441,-23.577,-43.674,179.818,5.752,149.075
C07930=1183.447,-23.846,-43.660,179.816,5.751,149.075
C07931=1183.452,-24.117,-43.647,179.813,5.751,149.076
C07932=1183.458,-24.366,-43.634,179.810,5.750,149.076
C07933=1183.463,-24.615,-43.622,179.808,5.750,149.077
C07934=1183.468,-24.865,-43.608,179.805,5.749,149.078
C07935=1183.473,-25.115,-43.596,179.803,5.749,149.078
C07936=1183.478,-25.364,-43.583,179.801,5.749,149.079
C07937=1183.484,-25.614,-43.571,179.798,5.749,149.080
C07938=1183.488,-25.864,-43.558,179.796,5.748,149.080
C07939=1183.493,-26.113,-43.545,179.793,5.747,149.081
C07940=1183.498,-26.363,-43.533,179.791,5.747,149.082
C07941=1183.503,-26.612,-43.520,179.788,5.746,149.082
C07942=1183.509,-26.862,-43.508,179.786,5.746,149.083
C07943=1183.513,-27.112,-43.495,179.784,5.746,149.083
C07944=1183.519,-27.362,-43.482,179.781,5.745,149.084
C07945=1183.524,-27.611,-43.470,179.779,5.745,149.085
C07946=1183.530,-27.861,-43.458,179.776,5.744,149.085
C07947=1183.535,-28.110,-43.445,179.774,5.744,149.086
C07948=1183.540,-28.359,-43.433,179.771,5.744,149.087
C07949=1183.545,-28.610,-43.420,179.769,5.743,149.087
C07950=1183.550,-28.859,-43.408,179.767,5.743,149.088
C07951=1183.555,-29.109,-43.395,179.764,5.742,149.089
C07952=1183.560,-29.358,-43.383,179.762,5.741,149.089
C07953=1183.566,-29.608,-43.371,179.759,5.741,149.090
C07954=1183.571,-29.857,-43.358,179.757,5.741,149.090
C07955=1183.575,-30.107,-43.345,179.754,5.741,149.091
C07956=1183.581,-30.357,-43.333,179.752,5.740,149.092
C07957=1183.586,-30.607,-43.321,179.750,5.740,149.092
C07958=1183.591,-30.856,-43.308,179.747,5.739,149.093
C07959=1183.596,-31.106,-43.296,179.745,5.740,149.094
C07960=1183.602,-31.355,-43.283,179.743,5.739,149.094
C07961=1183.607,-31.605,-43.272,179.740,5.738,149.095
C07962=1183.612,-31.855,-43.259,179.737,5.738,149.096
C07963=1183.617,-32.104,-43.246,179.735,5.737,149.096
C07964=1183.622,-32.354,-43.234,179.732,5.737,149.097
C07965=1183.627,-32.604,-43.222,179.730,5.737,149.097
C07966=1183.633,-32.854,-43.210,179.728,5.736,149.098
C07967=1183.638,-33.103,-43.197,179.726,5.736,149.099
C07968=1183.643,-33.352,-43.184,179.723,5.735,149.099
C07969=1183.648,-33.602,-43.173,179.720,5.735,149.100
C07970=1183.653,-33.852,-43.160,179.719,5.735,149.100
C07971=1183.659,-34.101,-43.148,179.716,5.734,149.101
C07972=1183.663,-34.351,-43.135,179.713,5.734,149.102
C07973=1183.669,-34.601,-43.123,179.711,5.733,149.103
C07974=1183.674,-34.851,-43.111,179.708,5.733,149.103
C07975=1183.679,-35.100,-43.099,179.706,5.733,149.104
C07976=1183.684,-35.350,-43.087,179.704,5.732,149.104
C07977=1183.689,-35.600,-43.075,179.702,5.732,149.105
C07978=1183.694,-35.849,-43.062,179.699,5.731,149.106
C07979=1183.700,-36.099,-43.050,179.696,5.731,149.106
C07980=1183.705,-36.348,-43.038,179.694,5.731,149.107
C07981=1183.710,-36.598,-43.026,179.692,5.730,149.107
C07982=1183.715,-36.847,-43.013,179.689,5.730,149.108
C07983=1183.721,-37.097,-43.001,179.687,5.729,149.109
C07984=1183.726,-37.347,-42.990,179.684,5.729,149.109
C07985=1183.731,-37.596,-42.978,179.682,5.729,149.110
C07986=1183.736,-37.846,-42.966,179.680,5.729,149.111
C07987=1183.741,-38.096,-42.953,179.677,5.728,149.111
C07988=1183.747,-38.346,-42.941,179.675,5.727,149.112
C07989=1183.752,-38.595,-42.929,179.672,5.727,149.113
C07990=1183.757,-38.845,-42.917,179.670,5.727,149.113
C07991=1183.763,-39.095,-42.905,179.668,5.726,149.114
C07992=1183.767,-39.344,-42.893,179.665,5.726,149.114
C07993=1183.772,-39.594,-42.881,179.663,5.725,149.115
C07994=1183.778,-39.844,-42.869,179.661,5.726,149.116
C07995=1183.783,-40.093,-42.856,179.658,5.725,149.116
C07996=1183.788,-40.343,-42.845,179.656,5.725,149.117
C07997=1183.793,-40.592,-42.833,179.653,5.724,149.118
C07998=1183.798,-40.842,-42.821,179.651,5.723,149.118
C07999=1183.804,-41.092,-42.809,179.649,5.724,149.119
C08000=1183.809,-41.341,-42.796,179.646,5.723,149.120
C08001=1183.814,-41.591,-42.784,179.644,5.722,149.120
C08002=1183.819,-41.841,-42.773,179.641,5.722,149.121
C08003=1183.824,-42.091,-42.761,179.639,5.722,149.121
C08004=1183.830,-42.340,-42.748,179.637,5.722,149.122
C08005=1183.835,-42.590,-42.737,179.634,5.721,149.123
C08006=1183.840,-42.839,-42.725,179.632,5.721,149.123
C08007=1183.845,-43.089,-42.713,179.630,5.721,149.124
C08008=1183.850,-43.339,-42.701,179.627,5.720,149.125
C08009=1183.856,-43.589,-42.689,179.625,5.720,149.125
C08010=1183.860,-43.838,-42.678,179.622,5.719,149.126
C08011=1183.865,-44.088,-42.665,179.619,5.719,149.127
C08012=1183.871,-44.337,-42.653,179.618,5.719,149.127
C08013=1183.876,-44.587,-42.642,179.615,5.718,149.128
C08014=1183.881,-44.837,-42.630,179.613,5.718,149.129
C08015=1183.886,-45.087,-42.618,179.610,5.717,149.129
C08016=1183.891,-45.336,-42.606,179.608,5.718,149.130
C08017=1183.896,-45.586,-42.594,179.606,5.717,149.130
C08018=1183.902,-45.836,-42.582,179.603,5.717,149.131
C08019=1183.908,-46.085,-42.571,179.601,5.716,149.132
C08020=1183.912,-46.335,-42.560,179.599,5.716,149.132
C08021=1183.917,-46.584,-42.547,179.596,5.716,149.133
C08022=1183.923,-46.834,-42.535,179.594,5.715,149.133
C08023=1183.928,-47.084,-42.524,179.591,5.715,149.134
C08024=1183.933,-47.334,-42.512,179.589,5.715,149.135
C08025=1183.938,-47.583,-42.500,179.587,5.714,149.135
C08026=1183.943,-47.833,-42.489,179.584,5.714,149.136
C08027=1183.949,-48.083,-42.477,179.582,5.713,149.137
C08028=1183.953,-48.333,-42.465,179.579,5.714,149.137
C08029=1183.959,-48.581,-42.453,179.577,5.713,149.138
C08030=1183.964,-48.831,-42.441,179.575,5.712,149.139
C08031=1183.969,-49.081,-42.430,179.572,5.712,149.139
C08032=1183.975,-49.352,-42.418,179.570,5.712,149.140
C08033=1183.981,-49.621,-42.405,179.568,5.711,149.140
C08034=1183.986,-49.892,-42.392,179.565,5.711,149.141
C08035=1183.991,-50.162,-42.379,179.562,5.711,149.142
C08036=1183.997,-50.412,-42.367,179.560,5.710,149.143
C08037=1184.002,-50.661,-42.356,179.557,5.710,149.143
C08038=1184.007,-50.911,-42.345,179.555,5.710,149.144
C08039=1184.013,-51.161,-42.333,179.553,5.709,149.144
C08040=1184.018,-51.411,-42.321,179.550,5.709,149.145
C08041=1184.023,-51.660,-42.310,179.548,5.709,149.146
C08042=1184.028,-51.910,-42.298,179.546,5.708,149.146
C08043=1184.034,-52.159,-42.287,179.543,5.708,149.147
C08044=1184.038,-52.409,-42.275,179.541,5.708,149.148
C08045=1184.044,-52.659,-42.264,179.539,5.707,149.148
C08046=1184.049,-52.909,-42.252,179.536,5.707,149.149
C08047=1184.054,-53.158,-42.240,179.534,5.707,149.150
C08048=1184.059,-53.408,-42.229,179.531,5.706,149.150
C08049=1184.065,-53.657,-42.218,179.529,5.706,149.151
C08050=1184.070,-53.907,-42.206,179.527,5.706,149.152
C08051=1184.075,-54.158,-42.195,179.524,5.705,149.152
C08052=1184.080,-54.407,-42.184,179.522,5.705,149.153
C08053=1184.085,-54.657,-42.172,179.520,5.705,149.153
C08054=1184.091,-54.906,-42.161,179.517,5.704,149.154
C08055=1184.096,-55.156,-42.149,179.515,5.704,149.155
C08056=1184.101,-55.406,-42.138,179.513,5.704,149.155
C08057=1184.106,-55.655,-42.126,179.510,5.704,149.156
C08058=1184.111,-55.905,-42.115,179.508,5.703,149.156
C08059=1184.117,-56.154,-42.103,179.506,5.703,149.157
C08060=1184.121,-56.404,-42.092,179.503,5.703,149.158
C08061=1184.127,-56.655,-42.081,179.501,5.702,149.158
C08062=1184.132,-56.904,-42.069,179.498,5.701,149.159
C08063=1184.138,-57.153,-42.058,179.496,5.702,149.160
C08064=1184.143,-57.403,-42.047,179.494,5.701,149.160
C08065=1184.147,-57.653,-42.035,179.491,5.701,149.161
C08066=1184.153,-57.903,-42.023,179.489,5.701,149.162
C08067=1184.158,-58.152,-42.012,179.487,5.701,149.162
C08068=1184.164,-58.402,-42.001,179.485,5.700,149.163
C08069=1184.168,-58.652,-41.990,179.482,5.700,149.164
C08070=1184.173,-58.901,-41.979,179.480,5.700,149.164
C08071=1184.179,-59.151,-41.967,179.478,5.699,149.165
C08072=1184.184,-59.400,-41.956,179.475,5.698,149.165
C08073=1184.190,-59.651,-41.945,179.473,5.699,149.166
C08074=1184.194,-59.900,-41.933,179.471,5.698,149.167
C08075=1184.200,-60.149,-41.923,179.468,5.698,149.167
C08076=1184.205,-60.399,-41.911,179.466,5.698,149.168
C08077=1184.210,-60.649,-41.900,179.464,5.697,149.169
C08078=1184.215,-60.898,-41.889,179.461,5.697,149.169
C08079=1184.221,-61.148,-41.877,179.459,5.697,149.170
C08080=1184.225,-61.398,-41.866,179.457,5.696,149.170
C08081=1184.231,-61.649,-41.855,179.454,5.696,149.171
C08082=1184.236,-61.897,-41.844,179.452,5.696,149.172
C08083=1184.241,-62.147,-41.833,179.450,5.695,149.172
C08084=1184.247,-62.398,-41.821,179.447,5.695,149.173
C08085=1184.252,-62.647,-41.811,179.445,5.695,149.174
C08086=1184.257,-62.896,-41.799,179.442,5.695,149.174
C08087=1184.262,-63.146,-41.787,179.440,5.694,149.175
C08088=1184.268,-63.396,-41.777,179.438,5.694,149.176
C08089=1184.273,-63.645,-41.766,179.436,5.694,149.176
C08090=1184.278,-63.896,-41.755,179.433,5.693,149.177
C08091=1184.284,-64.145,-41.744,179.431,5.693,149.177
C08092=1184.288,-64.394,-41.732,179.429,5.693,149.178
C08093=1184.293,-64.645,-41.722,179.426,5.692,149.179
C08094=1184.299,-64.894,-41.710,179.424,5.692,149.179
C08095=1184.304,-65.143,-41.699,179.422,5.692,149.180
C08096=1184.309,-65.394,-41.688,179.419,5.692,149.181
C08097=1184.314,-65.643,-41.678,179.417,5.691,149.181
C08098=1184.320,-65.893,-41.666,179.415,5.692,149.182
C08099=1184.325,-66.143,-41.655,179.413,5.691,149.182
C08100=1184.330,-66.392,-41.644,179.410,5.690,149.183
C08101=1184.335,-66.642,-41.634,179.408,5.691,149.184
C08102=1184.341,-66.891,-41.622,179.406,5.690,149.184
C08103=1184.346,-67.141,-41.612,179.403,5.690,149.185
C08104=1184.351,-67.391,-41.600,179.401,5.690,149.186
C08105=1184.356,-67.641,-41.590,179.399,5.689,149.186
C08106=1184.362,-67.891,-41.578,179.396,5.689,149.187
C08107=1184.367,-68.139,-41.567,179.394,5.689,149.188
C08108=1184.372,-68.390,-41.557,179.392,5.688,149.188
C08109=1184.377,-68.639,-41.545,179.389,5.688,149.189
C08110=1184.382,-68.889,-41.535,179.387,5.688,149.190
C08111=1184.388,-69.139,-41.523,179.385,5.687,149.190
C08112=1184.393,-69.388,-41.513,179.382,5.687,149.191
C08113=1184.398,-69.638,-41.502,179.380,5.687,149.191
C08114=1184.403,-69.888,-41.491,179.378,5.687,149.192
C08115=1184.408,-70.137,-41.480,179.375,5.686,149.193
C08116=1184.414,-70.388,-41.469,179.373,5.687,149.193
C08117=1184.420,-70.637,-41.459,179.371,5.686,149.194
C08118=1184.424,-70.887,-41.448,179.368,5.685,149.195
C08119=1184.430,-71.136,-41.437,179.366,5.686,149.195
C08120=1184.435,-71.386,-41.426,179.364,5.685,149.196
C08121=1184.440,-71.636,-41.416,179.361,5.684,149.196
C08122=1184.446,-71.886,-41.404,179.359,5.685,149.197
C08123=1184.451,-72.136,-41.393,179.357,5.684,149.198
C08124=1184.456,-72.385,-41.382,179.354,5.684,149.198
C08125=1184.461,-72.635,-41.372,179.352,5.684,149.199
C08126=1184.467,-72.885,-41.362,179.350,5.683,149.199
C08127=1184.471,-73.134,-41.350,179.348,5.684,149.200
C08128=1184.477,-73.384,-41.340,179.345,5.683,149.201
C08129=1184.482,-73.634,-41.330,179.343,5.682,149.201
C08130=1184.488,-73.883,-41.318,179.341,5.683,149.202
C08131=1184.493,-74.133,-41.308,179.338,5.682,149.203
C08132=1184.498,-74.382,-41.297,179.336,5.682,149.203
C08133=1184.503,-74.633,-41.286,179.334,5.682,149.204
C08134=1184.509,-74.882,-41.276,179.332,5.681,149.204
C08135=1184.514,-75.132,-41.265,179.329,5.681,149.205
C08136=1184.519,-75.403,-41.253,179.327,5.681,149.206
C08137=1184.525,-75.673,-41.242,179.325,5.681,149.207
C08138=1184.531,-75.945,-41.230,179.322,5.680,149.207
C08139=1184.536,-76.216,-41.218,179.319,5.680,149.208
C08140=1184.542,-76.465,-41.208,179.318,5.680,149.208
C08141=1184.548,-76.715,-41.198,179.315,5.679,149.209
C08142=1184.553,-76.965,-41.187,179.312,5.679,149.210
C08143=1184.558,-77.214,-41.176,179.311,5.679,149.210
C08144=1184.563,-77.464,-41.165,179.308,5.679,149.211
C08145=1184.569,-77.714,-41.155,179.306,5.679,149.212
C08146=1184.573,-77.964,-41.144,179.304,5.678,149.212
C08147=1184.579,-78.213,-41.134,179.301,5.678,149.213
C08148=1184.584,-78.463,-41.123,179.299,5.678,149.213
C08149=1184.589,-78.713,-41.113,179.297,5.677,149.214
C08150=1184.594,-78.963,-41.102,179.294,5.677,149.215
C08151=1184.600,-79.212,-41.091,179.293,5.677,149.215
C08152=1184.605,-79.462,-41.081,179.290,5.677,149.216
C08153=1184.610,-79.712,-41.071,179.288,5.677,149.217
C08154=1184.616,-79.961,-41.060,179.286,5.676,149.217
C08155=1184.621,-80.211,-41.049,179.283,5.676,149.218
C08156=1184.626,-80.461,-41.039,179.281,5.676,149.219
C08157=1184.631,-80.711,-41.028,179.279,5.675,149.219
C08158=1184.637,-80.960,-41.018,179.276,5.675,149.220
C08159=1184.642,-81.211,-41.008,179.274,5.675,149.220
C08160=1184.647,-81.460,-40.997,179.272,5.675,149.221
C08161=1184.653,-81.709,-40.986,179.270,5.675,149.222
C08162=1184.657,-81.959,-40.976,179.267,5.674,149.222
C08163=1184.663,-82.209,-40.966,179.265,5.674,149.223
C08164=1184.668,-82.459,-40.956,179.263,5.674,149.224
C08165=1184.673,-82.708,-40.945,179.260,5.673,149.224
C08166=1184.678,-82.959,-40.935,179.258,5.674,149.225
C08167=1184.684,-83.208,-40.925,179.256,5.673,149.225
C08168=1184.689,-83.458,-40.915,179.254,5.672,149.226
C08169=1184.694,-83.707,-40.903,179.251,5.673,149.227
C08170=1184.700,-83.957,-40.893,179.249,5.672,149.227
C08171=1184.705,-84.207,-40.882,179.247,5.672,149.228
C08172=1184.710,-84.457,-40.872,179.245,5.672,149.229
C08173=1184.715,-84.706,-40.863,179.242,5.671,149.229
C08174=1184.720,-84.956,-40.852,179.240,5.672,149.230
C08175=1184.726,-85.206,-40.842,179.238,5.671,149.230
C08176=1184.731,-85.455,-40.832,179.236,5.671,149.231
C08177=1184.736,-85.705,-40.821,179.233,5.671,149.232
C08178=1184.742,-85.955,-40.811,179.231,5.670,149.232
C08179=1184.747,-86.205,-40.800,179.229,5.670,149.233
C08180=1184.752,-86.454,-40.791,179.226,5.670,149.234
C08181=1184.757,-86.704,-40.780,179.225,5.670,149.234
C08182=1184.762,-86.954,-40.770,179.222,5.670,149.235
C08183=1184.768,-87.204,-40.760,179.220,5.669,149.235
C08184=1184.774,-87.453,-40.749,179.218,5.669,149.236
C08185=1184.779,-87.704,-40.739,179.215,5.669,149.237
C08186=1184.783,-87.953,-40.729,179.214,5.669,149.237
C08187=1184.789,-88.202,-40.719,179.211,5.668,149.238
C08188=1184.794,-88.453,-40.708,179.208,5.668,149.239
C08189=1184.800,-88.702,-40.698,179.207,5.668,149.239
C08190=1184.805,-88.952,-40.688,179.204,5.668,149.240
C08191=1184.809,-89.202,-40.678,179.202,5.668,149.240
C08192=1184.815,-89.451,-40.668,179.200,5.667,149.241
C08193=1184.821,-89.701,-40.658,179.197,5.667,149.242
C08194=1184.826,-89.951,-40.647,179.195,5.667,149.242
C08195=1184.830,-90.200,-40.637,179.193,5.666,149.243
C08196=1184.836,-90.450,-40.627,179.191,5.666,149.243
C08197=1184.841,-90.701,-40.617,179.188,5.666,149.244
C08198=1184.847,-90.950,-40.607,179.186,5.666,149.245
C08199=1184.852,-91.199,-40.598,179.184,5.666,149.245
C08200=1184.857,-91.449,-40.587,179.181,5.665,149.246
C08201=1184.862,-91.699,-40.577,179.180,5.665,149.247
C08202=1184.868,-91.949,-40.567,179.177,5.665,149.247
C08203=1184.873,-92.198,-40.557,179.175,5.665,149.248
C08204=1184.878,-92.448,-40.546,179.173,5.664,149.248
C08205=1184.884,-92.698,-40.537,179.171,5.665,149.249
C08206=1184.889,-92.948,-40.527,179.169,5.664,149.250
C08207=1184.894,-93.197,-40.517,179.166,5.664,149.250
C08208=1184.899,-93.447,-40.507,179.164,5.664,149.251
C08209=1184.905,-93.697,-40.496,179.162,5.663,149.252
C08210=1184.910,-93.946,-40.487,179.160,5.664,149.252
C08211=1184.916,-94.196,-40.477,179.157,5.663,149.253
C08212=1184.921,-94.447,-40.467,179.155,5.663,149.253
C08213=1184.926,-94.696,-40.456,179.153,5.663,149.254
C08214=1184.931,-94.945,-40.447,179.151,5.662,149.255
C08215=1184.937,-95.195,-40.437,179.148,5.662,149.255
C08216=1184.942,-95.446,-40.427,179.146,5.662,149.256
C08217=1184.947,-95.695,-40.417,179.144,5.662,149.257
C08218=1184.952,-95.945,-40.407,179.142,5.661,149.257
C08219=1184.958,-96.194,-40.397,179.140,5.662,149.258
C08220=1184.963,-96.444,-40.388,179.137,5.661,149.258
C08221=1184.968,-96.694,-40.377,179.135,5.660,149.259
C08222=1184.973,-96.943,-40.368,179.133,5.661,149.260
C08223=1184.979,-97.193,-40.357,179.131,5.660,149.260
C08224=1184.985,-97.443,-40.348,179.129,5.660,149.261
C08225=1184.989,-97.693,-40.338,179.126,5.660,149.262
C08226=1184.994,-97.943,-40.328,179.124,5.660,149.262
C08227=1185.000,-98.193,-40.318,179.122,5.660,149.263
C08228=1185.005,-98.442,-40.309,179.120,5.660,149.263
C08229=1185.011,-98.691,-40.298,179.117,5.659,149.264
C08230=1185.017,-98.942,-40.289,179.115,5.659,149.264
C08231=1185.021,-99.192,-40.279,179.113,5.659,149.265
C08232=1185.027,-99.441,-40.269,179.110,5.659,149.266
C08233=1185.032,-99.691,-40.260,179.109,5.659,149.266
C08234=1185.037,-99.941,-40.250,179.106,5.658,149.267
C08235=1185.042,-100.190,-40.240,179.105,5.658,149.268
C08236=1185.047,-100.441,-40.230,179.102,5.658,149.268
C08237=1185.053,-100.690,-40.220,179.100,5.658,149.269
C08238=1185.058,-100.939,-40.210,179.098,5.657,149.269
C08239=1185.064,-101.190,-40.201,179.095,5.657,149.270
C08240=1185.069,-101.461,-40.190,179.093,5.657,149.271
C08241=1185.075,-101.733,-40.180,179.091,5.657,149.271
C08242=1185.081,-102.004,-40.169,179.088,5.656,149.272
C08243=1185.087,-102.276,-40.158,179.086,5.657,149.273
C08244=1185.092,-102.525,-40.149,179.084,5.656,149.273
C08245=1185.097,-102.775,-40.139,179.082,5.656,149.274
C08246=1185.102,-103.026,-40.130,179.079,5.655,149.274
C08247=1185.107,-103.275,-40.120,179.077,5.656,149.275
C08248=1185.112,-103.524,-40.110,179.075,5.655,149.276
C08249=1185.118,-103.774,-40.101,179.073,5.655,149.276
C08250=1185.123,-104.024,-40.091,179.070,5.655,149.277
C08251=1185.129,-104.274,-40.081,179.068,5.654,149.278
C08252=1185.134,-104.523,-40.072,179.066,5.655,149.278
C08253=1185.140,-104.773,-40.062,179.064,5.654,149.279
C08254=1185.144,-105.023,-40.052,179.062,5.654,149.279
C08255=1185.150,-105.273,-40.043,179.060,5.654,149.280
C08256=1185.155,-105.523,-40.033,179.058,5.654,149.281
C08257=1185.161,-105.773,-40.024,179.055,5.654,149.281
C08258=1185.166,-106.022,-40.014,179.053,5.654,149.282
C08259=1185.171,-106.272,-40.005,179.051,5.653,149.283
C08260=1185.176,-106.521,-39.995,179.049,5.653,149.283
C08261=1185.182,-106.772,-39.986,179.046,5.653,149.284
C08262=1185.187,-107.021,-39.976,179.045,5.653,149.284
C08263=1185.192,-107.271,-39.967,179.042,5.652,149.285
C08264=1185.197,-107.521,-39.956,179.041,5.652,149.285
C08265=1185.202,-107.771,-39.948,179.038,5.652,149.286
C08266=1185.208,-108.020,-39.937,179.036,5.651,149.287
C08267=1185.213,-108.270,-39.928,179.034,5.652,149.287
C08268=1185.219,-108.520,-39.919,179.031,5.651,149.288
C08269=1185.224,-108.770,-39.909,179.029,5.651,149.289
C08270=1185.229,-109.019,-39.900,179.027,5.651,149.289
C08271=1185.235,-109.269,-39.890,179.025,5.651,149.290
C08272=1185.240,-109.519,-39.881,179.022,5.650,149.291
C08273=1185.246,-109.769,-39.872,179.021,5.651,149.291
C08274=1185.251,-110.018,-39.862,179.018,5.650,149.292
C08275=1185.256,-110.268,-39.853,179.016,5.650,149.292
C08276=1185.261,-110.518,-39.843,179.014,5.650,149.293
C08277=1185.267,-110.767,-39.834,179.012,5.650,149.293
C08278=1185.272,-111.018,-39.825,179.010,5.649,149.294
C08279=1185.277,-111.267,-39.815,179.008,5.649,149.295
C08280=1185.282,-111.517,-39.806,179.005,5.649,149.295
C08281=1185.288,-111.767,-39.797,179.004,5.649,149.296
C08282=1185.293,-112.016,-39.787,179.001,5.649,149.297
C08283=1185.298,-112.266,-39.778,178.999,5.649,149.297
C08284=1185.304,-112.516,-39.769,178.997,5.648,149.298
C08285=1185.309,-112.765,-39.759,178.995,5.648,149.298
C08286=1185.314,-113.015,-39.750,178.992,5.648,149.299
C08287=1185.320,-113.265,-39.741,178.990,5.648,149.300
C08288=1185.325,-113.515,-39.731,178.988,5.648,149.300
C08289=1185.330,-113.764,-39.722,178.986,5.648,149.301
C08290=1185.336,-114.015,-39.713,178.984,5.647,149.301
C08291=1185.341,-114.264,-39.704,178.982,5.648,149.302
C08292=1185.346,-114.514,-39.694,178.980,5.647,149.303
C08293=1185.352,-114.764,-39.685,178.978,5.647,149.303
C08294=1185.357,-115.014,-39.676,178.975,5.646,149.304
C08295=1185.362,-115.264,-39.667,178.973,5.647,149.304
C08296=1185.367,-115.513,-39.657,178.971,5.646,149.305
C08297=1185.373,-115.763,-39.648,178.969,5.646,149.306
C08298=1185.378,-116.013,-39.639,178.967,5.646,149.306
C08299=1185.384,-116.263,-39.630,178.965,5.646,149.307
C08300=1185.389,-116.512,-39.620,178.962,5.645,149.307
C08301=1185.394,-116.762,-39.611,178.960,5.646,149.308
C08302=1185.399,-117.012,-39.602,178.958,5.645,149.309
C08303=1185.405,-117.262,-39.593,178.956,5.645,149.309
C08304=1185.411,-117.512,-39.584,178.954,5.645,149.310
C08305=1185.415,-117.761,-39.574,178.952,5.645,149.310
C08306=1185.421,-118.011,-39.565,178.950,5.644,149.311
C08307=1185.426,-118.261,-39.556,178.948,5.645,149.312
C08308=1185.432,-118.511,-39.547,178.945,5.644,149.312
C08309=1185.437,-118.761,-39.538,178.943,5.644,149.313
C08310=1185.442,-119.011,-39.529,178.941,5.643,149.313
C08311=1185.447,-119.260,-39.519,178.939,5.644,149.314
C08312=1185.452,-119.510,-39.510,178.937,5.643,149.315
C08313=1185.459,-119.759,-39.501,178.935,5.644,149.315
C08314=1185.464,-120.009,-39.492,178.933,5.643,149.316
C08315=1185.469,-120.259,-39.484,178.930,5.643,149.316
C08316=1185.474,-120.509,-39.475,178.928,5.642,149.317
C08317=1185.479,-120.759,-39.466,178.926,5.643,149.318
C08318=1185.485,-121.009,-39.456,178.924,5.642,149.318
C08319=1185.490,-121.259,-39.447,178.922,5.642,149.319
C08320=1185.495,-121.508,-39.438,178.920,5.642,149.319
C08321=1185.500,-121.758,-39.429,178.918,5.642,149.320
C08322=1185.505,-122.008,-39.420,178.915,5.641,149.321
C08323=1185.511,-122.257,-39.411,178.914,5.641,149.321
C08324=1185.517,-122.507,-39.402,178.911,5.641,149.322
C08325=1185.522,-122.757,-39.393,178.910,5.641,149.322
C08326=1185.527,-123.007,-39.384,178.907,5.641,149.323
C08327=1185.533,-123.256,-39.375,178.905,5.641,149.323
C08328=1185.538,-123.506,-39.366,178.903,5.640,149.324
C08329=1185.543,-123.756,-39.357,178.901,5.640,149.325
C08330=1185.548,-124.006,-39.349,178.898,5.640,149.325
C08331=1185.553,-124.256,-39.340,178.897,5.640,149.326
C08332=1185.560,-124.505,-39.330,178.894,5.639,149.327
C08333=1185.565,-124.755,-39.322,178.892,5.639,149.327
C08334=1185.570,-125.005,-39.313,178.890,5.639,149.328
C08335=1185.575,-125.255,-39.304,178.888,5.639,149.328
C08336=1185.580,-125.505,-39.295,178.886,5.638,149.329
C08337=1185.586,-125.755,-39.286,178.884,5.639,149.329
C08338=1185.591,-126.004,-39.277,178.882,5.638,149.330
C08339=1185.597,-126.254,-39.269,178.880,5.638,149.331
C08340=1185.602,-126.503,-39.260,178.878,5.638,149.331
C08341=1185.607,-126.753,-39.251,178.875,5.638,149.332
C08342=1185.613,-127.003,-39.241,178.874,5.638,149.332
C08343=1185.618,-127.253,-39.232,178.871,5.638,149.333
C08344=1185.197,-127.264,-39.273,178.867,5.641,149.335
C08345=1185.191,-127.015,-39.281,178.870,5.641,149.334
C08346=1185.186,-126.765,-39.290,178.871,5.641,149.334
C08347=1185.181,-126.515,-39.299,178.874,5.642,149.333
C08348=1185.176,-126.265,-39.308,178.876,5.642,149.333
C08349=1185.170,-126.015,-39.317,178.878,5.642,149.332
C08350=1185.165,-125.765,-39.325,178.880,5.642,149.331
C08351=1185.158,-125.515,-39.334,178.882,5.643,149.331
C08352=1185.153,-125.266,-39.343,178.884,5.642,149.330
C08353=1185.148,-125.016,-39.352,178.886,5.643,149.330
C08354=1185.143,-124.766,-39.361,178.889,5.643,149.329
C08355=1185.138,-124.516,-39.370,178.890,5.643,149.328
C08356=1185.133,-124.266,-39.379,178.893,5.643,149.328
C08357=1185.127,-124.016,-39.388,178.894,5.643,149.327
C08358=1185.122,-123.767,-39.396,178.897,5.643,149.326
C08359=1185.116,-123.517,-39.405,178.899,5.643,149.326
C08360=1185.111,-123.268,-39.415,178.901,5.644,149.325
C08361=1185.106,-123.018,-39.424,178.903,5.644,149.325
C08362=1185.101,-122.768,-39.433,178.905,5.645,149.324
C08363=1185.095,-122.518,-39.442,178.907,5.644,149.324
C08364=1185.090,-122.268,-39.451,178.909,5.645,149.323
C08365=1185.085,-122.018,-39.460,178.912,5.644,149.322
C08366=1185.080,-121.769,-39.469,178.914,5.645,149.322
C08367=1185.073,-121.519,-39.478,178.916,5.645,149.321
C08368=1185.068,-121.269,-39.487,178.918,5.646,149.321
C08369=1185.063,-121.019,-39.496,178.920,5.645,149.320
C08370=1185.058,-120.770,-39.504,178.922,5.646,149.319
C08371=1185.053,-120.520,-39.513,178.924,5.646,149.319
C08372=1185.048,-120.270,-39.522,178.927,5.646,149.318
C08373=1185.042,-120.020,-39.532,178.929,5.646,149.318
C08374=1185.037,-119.770,-39.541,178.931,5.647,149.317
C08375=1185.032,-119.521,-39.550,178.933,5.646,149.316
C08376=1185.026,-119.271,-39.559,178.935,5.647,149.316
C08377=1185.021,-119.021,-39.568,178.937,5.647,149.315
C08378=1185.015,-118.771,-39.578,178.939,5.647,149.315
C08379=1185.010,-118.522,-39.586,178.941,5.647,149.314
C08380=1185.005,-118.272,-39.596,178.944,5.648,149.313
C08381=1185.000,-118.023,-39.605,178.946,5.647,149.313
C08382=1184.994,-117.772,-39.614,178.948,5.648,149.312
C08383=1184.989,-117.523,-39.623,178.950,5.648,149.312
C08384=1184.983,-117.273,-39.632,178.952,5.649,149.311
C08385=1184.978,-117.023,-39.641,178.954,5.648,149.310
C08386=1184.973,-116.773,-39.651,178.956,5.649,149.310
C08387=1184.967,-116.523,-39.660,178.959,5.648,149.309
C08388=1184.962,-116.274,-39.669,178.961,5.649,149.309
C08389=1184.957,-116.024,-39.678,178.963,5.649,149.308
C08390=1184.952,-115.774,-39.688,178.965,5.650,149.307
C08391=1184.946,-115.524,-39.697,178.967,5.649,149.307
C08392=1184.941,-115.274,-39.706,178.969,5.650,149.306
C08393=1184.935,-115.024,-39.715,178.971,5.650,149.306
C08394=1184.930,-114.774,-39.724,178.974,5.650,149.305
C08395=1184.925,-114.525,-39.734,178.976,5.650,149.304
C08396=1184.920,-114.275,-39.743,178.978,5.651,149.304
C08397=1184.914,-114.025,-39.752,178.980,5.650,149.303
C08398=1184.909,-113.776,-39.762,178.982,5.651,149.303
C08399=1184.904,-113.526,-39.771,178.984,5.651,149.302
C08400=1184.898,-113.276,-39.780,178.986,5.651,149.301
C08401=1184.893,-113.026,-39.789,178.989,5.651,149.301
C08402=1184.888,-112.777,-39.799,178.991,5.652,149.300
C08403=1184.882,-112.527,-39.808,178.993,5.651,149.300
C08404=1184.877,-112.277,-39.817,178.995,5.652,149.299
C08405=1184.872,-112.028,-39.827,178.997,5.652,149.298
C08406=1184.866,-111.777,-39.836,178.999,5.653,149.298
C08407=1184.861,-111.528,-39.845,179.001,5.652,149.297
C08408=1184.856,-111.278,-39.855,179.004,5.653,149.297
C08409=1184.850,-111.028,-39.864,179.006,5.653,149.296
C08410=1184.845,-110.778,-39.873,179.008,5.653,149.295
C08411=1184.840,-110.529,-39.883,179.010,5.653,149.295
C08412=1184.835,-110.279,-39.892,179.012,5.654,149.294
C08413=1184.829,-110.029,-39.901,179.014,5.653,149.294
C08414=1184.824,-109.780,-39.911,179.016,5.654,149.293
C08415=1184.819,-109.530,-39.920,179.019,5.654,149.292
C08416=1184.814,-109.281,-39.930,179.021,5.654,149.292
C08417=1184.808,-109.030,-39.939,179.023,5.655,149.291
C08418=1184.803,-108.781,-39.948,179.025,5.654,149.290
C08419=1184.797,-108.531,-39.958,179.028,5.655,149.290
C08420=1184.792,-108.281,-39.967,179.030,5.655,149.289
C08421=1184.786,-108.032,-39.977,179.032,5.656,149.289
C08422=1184.781,-107.782,-39.986,179.034,5.655,149.288
C08423=1184.777,-107.532,-39.996,179.036,5.656,149.288
C08424=1184.771,-107.282,-40.006,179.038,5.656,149.287
C08425=1184.766,-107.032,-40.015,179.040,5.656,149.286
C08426=1184.760,-106.782,-40.025,179.042,5.656,149.286
C08427=1184.755,-106.532,-40.034,179.045,5.657,149.285
C08428=1184.749,-106.283,-40.044,179.047,5.656,149.284
C08429=1184.744,-106.033,-40.053,179.049,5.657,149.284
C08430=1184.739,-105.784,-40.063,179.051,5.657,149.283
C08431=1184.733,-105.534,-40.072,179.054,5.657,149.283
C08432=1184.729,-105.284,-40.082,179.055,5.657,149.282
C08433=1184.723,-105.034,-40.091,179.058,5.657,149.281
C08434=1184.718,-104.784,-40.101,179.060,5.658,149.281
C08435=1184.713,-104.534,-40.111,179.062,5.658,149.280
C08436=1184.708,-104.285,-40.120,179.064,5.659,149.280
C08437=1184.702,-104.035,-40.130,179.067,5.658,149.279
C08438=1184.697,-103.785,-40.139,179.069,5.659,149.278
C08439=1184.691,-103.536,-40.150,179.071,5.659,149.278
C08440=1184.686,-103.286,-40.158,179.074,5.659,149.277
C08441=1184.681,-103.037,-40.169,179.075,5.659,149.277
C08442=1184.676,-102.786,-40.178,179.078,5.659,149.276
C08443=1184.670,-102.536,-40.188,179.079,5.659,149.275
C08444=1184.665,-102.287,-40.197,179.082,5.660,149.275
C08445=1184.659,-102.015,-40.209,179.085,5.660,149.274
C08446=1184.653,-101.744,-40.218,179.086,5.660,149.273
C08447=1184.648,-101.472,-40.229,179.089,5.661,149.273
C08448=1184.642,-101.200,-40.240,179.092,5.661,149.272
C08449=1184.637,-100.950,-40.249,179.093,5.661,149.272
C08450=1184.631,-100.701,-40.259,179.096,5.661,149.271
C08451=1184.626,-100.452,-40.269,179.098,5.661,149.270
C08452=1184.621,-100.201,-40.279,179.100,5.662,149.270
C08453=1184.616,-99.951,-40.288,179.102,5.661,149.269
C08454=1184.610,-99.702,-40.299,179.105,5.662,149.268
C08455=1184.605,-99.452,-40.307,179.107,5.663,149.268
C08456=1184.600,-99.203,-40.318,179.109,5.663,149.267
C08457=1184.595,-98.952,-40.328,179.111,5.663,149.267
C08458=1184.589,-98.702,-40.337,179.114,5.662,149.266
C08459=1184.584,-98.453,-40.347,179.116,5.663,149.265
C08460=1184.579,-98.204,-40.357,179.118,5.663,149.265
C08461=1184.573,-97.954,-40.366,179.120,5.664,149.264
C08462=1184.568,-97.704,-40.377,179.122,5.663,149.263
C08463=1184.563,-97.454,-40.387,179.124,5.664,149.263
C08464=1184.557,-97.204,-40.396,179.127,5.664,149.262
C08465=1184.552,-96.954,-40.406,179.129,5.664,149.262
C08466=1184.547,-96.705,-40.416,179.131,5.665,149.261
C08467=1184.542,-96.455,-40.427,179.133,5.664,149.260
C08468=1184.536,-96.205,-40.436,179.136,5.665,149.260
C08469=1184.531,-95.955,-40.446,179.138,5.665,149.259
C08470=1184.526,-95.706,-40.456,179.140,5.666,149.259
C08471=1184.520,-95.456,-40.466,179.142,5.665,149.258
C08472=1184.515,-95.206,-40.475,179.145,5.666,149.257
C08473=1184.510,-94.956,-40.486,179.147,5.666,149.257
C08474=1184.504,-94.707,-40.496,179.149,5.666,149.256
C08475=1184.499,-94.458,-40.505,179.151,5.667,149.256
C08476=1184.494,-94.207,-40.515,179.153,5.666,149.255
C08477=1184.488,-93.957,-40.525,179.156,5.667,149.254
C08478=1184.484,-93.708,-40.535,179.157,5.667,149.254
C08479=1184.478,-93.458,-40.545,179.160,5.667,149.253
C08480=1184.473,-93.208,-40.556,179.162,5.668,149.252
C08481=1184.468,-92.959,-40.565,179.164,5.668,149.252
C08482=1184.462,-92.709,-40.575,179.167,5.668,149.251
C08483=1184.457,-92.459,-40.585,179.169,5.668,149.251
C08484=1184.452,-92.209,-40.596,179.171,5.668,149.250
C08485=1184.447,-91.960,-40.605,179.173,5.669,149.249
C08486=1184.441,-91.710,-40.616,179.176,5.669,149.249
C08487=1184.436,-91.460,-40.626,179.178,5.669,149.248
C08488=1184.431,-91.210,-40.636,179.180,5.669,149.247
C08489=1184.425,-90.960,-40.645,179.182,5.670,149.247
C08490=1184.420,-90.711,-40.655,179.184,5.670,149.246
C08491=1184.415,-90.461,-40.666,179.187,5.670,149.246
C08492=1184.409,-90.211,-40.676,179.189,5.670,149.245
C08493=1184.404,-89.962,-40.686,179.191,5.670,149.244
C08494=1184.399,-89.712,-40.696,179.194,5.671,149.244
C08495=1184.394,-89.462,-40.707,179.195,5.671,149.243
C08496=1184.388,-89.213,-40.717,179.198,5.671,149.242
C08497=1184.384,-88.963,-40.727,179.201,5.672,149.242
C08498=1184.378,-88.713,-40.737,179.202,5.672,149.241
C08499=1184.373,-88.464,-40.747,179.205,5.672,149.241
C08500=1184.368,-88.213,-40.758,179.206,5.672,149.240
C08501=1184.362,-87.964,-40.768,179.209,5.672,149.239
C08502=1184.357,-87.715,-40.778,179.211,5.672,149.239
C08503=1184.352,-87.464,-40.788,179.213,5.673,149.238
C08504=1184.347,-87.215,-40.798,179.216,5.673,149.237
C08505=1184.341,-86.965,-40.809,179.218,5.673,149.237
C08506=1184.336,-86.715,-40.819,179.220,5.674,149.236
C08507=1184.330,-86.465,-40.829,179.222,5.673,149.236
C08508=1184.326,-86.216,-40.839,179.225,5.674,149.235
C08509=1184.321,-85.966,-40.850,179.227,5.674,149.234
C08510=1184.315,-85.716,-40.860,179.229,5.674,149.234
C08511=1184.309,-85.467,-40.870,179.232,5.675,149.233
C08512=1184.304,-85.217,-40.881,179.234,5.674,149.232
C08513=1184.299,-84.967,-40.891,179.236,5.675,149.232
C08514=1184.294,-84.717,-40.901,179.239,5.676,149.231
C08515=1184.289,-84.468,-40.911,179.241,5.675,149.231
C08516=1184.283,-84.218,-40.921,179.243,5.676,149.230
C08517=1184.278,-83.968,-40.932,179.245,5.676,149.229
C08518=1184.273,-83.718,-40.942,179.247,5.676,149.229
C08519=1184.267,-83.469,-40.952,179.250,5.677,149.228
C08520=1184.262,-83.218,-40.963,179.252,5.676,149.227
C08521=1184.257,-82.969,-40.973,179.254,5.677,149.227
C08522=1184.252,-82.719,-40.984,179.256,5.677,149.226
C08523=1184.246,-82.470,-40.994,179.259,5.677,149.226
C08524=1184.242,-82.220,-41.004,179.261,5.678,149.225
C08525=1184.236,-81.970,-41.015,179.263,5.678,149.224
C08526=1184.231,-81.721,-41.025,179.265,5.678,149.224
C08527=1184.226,-81.471,-41.035,179.268,5.679,149.223
C08528=1184.220,-81.221,-41.046,179.270,5.678,149.222
C08529=1184.216,-80.971,-41.057,179.272,5.679,149.222
C08530=1184.210,-80.722,-41.067,179.274,5.679,149.221
C08531=1184.204,-80.472,-41.077,179.277,5.679,149.221
C08532=1184.199,-80.222,-41.088,179.279,5.680,149.220
C08533=1184.194,-79.972,-41.098,179.281,5.680,149.219
C08534=1184.189,-79.722,-41.109,179.284,5.680,149.219
C08535=1184.183,-79.473,-41.120,179.285,5.680,149.218
C08536=1184.178,-79.223,-41.130,179.288,5.681,149.217
C08537=1184.173,-78.974,-41.140,179.290,5.681,149.217
C08538=1184.168,-78.723,-41.151,179.292,5.681,149.216
C08539=1184.162,-78.474,-41.161,179.295,5.681,149.216
C08540=1184.157,-78.225,-41.172,179.297,5.682,149.215
C08541=1184.152,-77.975,-41.183,179.299,5.682,149.214
C08542=1184.146,-77.725,-41.193,179.302,5.682,149.214
C08543=1184.141,-77.475,-41.203,179.304,5.682,149.213
C08544=1184.136,-77.226,-41.214,179.306,5.683,149.212
C08545=1184.131,-76.976,-41.225,179.309,5.683,149.212
C08546=1184.125,-76.726,-41.235,179.311,5.683,149.211
C08547=1184.121,-76.476,-41.246,179.313,5.683,149.211
C08548=1184.115,-76.227,-41.257,179.315,5.684,149.210
C08549=1184.109,-75.955,-41.268,179.317,5.684,149.209
C08550=1184.104,-75.685,-41.280,179.320,5.684,149.209
C08551=1184.098,-75.414,-41.291,179.323,5.685,149.208
C08552=1184.092,-75.143,-41.303,179.325,5.685,149.207
C08553=1184.087,-74.893,-41.314,179.328,5.685,149.207
C08554=1184.082,-74.644,-41.325,179.330,5.685,149.206
C08555=1184.076,-74.394,-41.335,179.332,5.686,149.205
C08556=1184.071,-74.144,-41.346,179.335,5.685,149.205
C08557=1184.066,-73.895,-41.356,179.337,5.686,149.204
C08558=1184.061,-73.645,-41.367,179.339,5.687,149.203
C08559=1184.055,-73.395,-41.377,179.341,5.686,149.203
C08560=1184.050,-73.145,-41.389,179.344,5.687,149.202
C08561=1184.044,-72.896,-41.399,179.346,5.688,149.202
C08562=1184.039,-72.645,-41.410,179.348,5.688,149.201
C08563=1184.035,-72.396,-41.421,179.351,5.688,149.200
C08564=1184.029,-72.146,-41.431,179.353,5.688,149.200
C08565=1184.024,-71.897,-41.443,179.355,5.688,149.199
C08566=1184.019,-71.647,-41.453,179.358,5.689,149.198
C08567=1184.014,-71.397,-41.464,179.360,5.688,149.198
C08568=1184.008,-71.148,-41.475,179.362,5.689,149.197
C08569=1184.003,-70.897,-41.486,179.364,5.690,149.197
C08570=1183.998,-70.648,-41.497,179.367,5.689,149.196
C08571=1183.993,-70.398,-41.507,179.369,5.690,149.195
C08572=1183.988,-70.148,-41.518,179.371,5.690,149.195
C08573=1183.982,-69.899,-41.529,179.373,5.690,149.194
C08574=1183.977,-69.649,-41.540,179.376,5.691,149.194
C08575=1183.971,-69.399,-41.551,179.378,5.691,149.193
C08576=1183.967,-69.150,-41.562,179.380,5.691,149.192
C08577=1183.961,-68.900,-41.572,179.383,5.692,149.192
C08578=1183.956,-68.651,-41.583,179.385,5.692,149.191
C08579=1183.950,-68.400,-41.595,179.387,5.692,149.190
C08580=1183.945,-68.151,-41.606,179.390,5.693,149.190
C08581=1183.940,-67.901,-41.616,179.392,5.693,149.189
C08582=1183.935,-67.652,-41.627,179.394,5.693,149.188
C08583=1183.929,-67.401,-41.638,179.396,5.693,149.188
C08584=1183.924,-67.152,-41.650,179.399,5.694,149.187
C08585=1183.919,-66.902,-41.660,179.401,5.693,149.186
C08586=1183.914,-66.653,-41.671,179.403,5.694,149.186
C08587=1183.909,-66.403,-41.682,179.406,5.695,149.185
C08588=1183.903,-66.153,-41.693,179.408,5.694,149.185
C08589=1183.898,-65.904,-41.704,179.410,5.695,149.184
C08590=1183.893,-65.654,-41.715,179.413,5.696,149.183
C08591=1183.888,-65.404,-41.726,179.415,5.695,149.183
C08592=1183.883,-65.154,-41.738,179.417,5.696,149.182
C08593=1183.877,-64.905,-41.748,179.420,5.696,149.181
C08594=1183.872,-64.655,-41.759,179.422,5.696,149.181
C08595=1183.867,-64.405,-41.770,179.424,5.697,149.180
C08596=1183.861,-64.156,-41.781,179.427,5.697,149.180
C08597=1183.857,-63.906,-41.793,179.429,5.697,149.179
C08598=1183.852,-63.656,-41.803,179.431,5.698,149.178
C08599=1183.846,-63.407,-41.815,179.434,5.698,149.178
C08600=1183.841,-63.157,-41.826,179.436,5.698,149.177
C08601=1183.836,-62.907,-41.837,179.438,5.699,149.176
C08602=1183.830,-62.658,-41.848,179.441,5.699,149.176
C08603=1183.825,-62.408,-41.859,179.443,5.699,149.175
C08604=1183.820,-62.158,-41.870,179.445,5.699,149.175
C08605=1183.814,-61.908,-41.882,179.448,5.700,149.174
C08606=1183.810,-61.659,-41.893,179.450,5.700,149.173
C08607=1183.805,-61.409,-41.904,179.452,5.700,149.173
C08608=1183.799,-61.159,-41.915,179.455,5.701,149.172
C08609=1183.794,-60.910,-41.926,179.457,5.701,149.171
C08610=1183.789,-60.660,-41.938,179.459,5.701,149.171
C08611=1183.783,-60.410,-41.949,179.462,5.701,149.170
C08612=1183.778,-60.161,-41.960,179.464,5.702,149.169
C08613=1183.773,-59.911,-41.972,179.466,5.702,149.169
C08614=1183.768,-59.661,-41.983,179.468,5.702,149.168
C08615=1183.763,-59.412,-41.994,179.471,5.703,149.168
C08616=1183.757,-59.162,-42.005,179.474,5.703,149.167
C08617=1183.752,-58.912,-42.016,179.475,5.703,149.166
C08618=1183.748,-58.662,-42.027,179.478,5.704,149.166
C08619=1183.742,-58.413,-42.039,179.481,5.704,149.165
C08620=1183.737,-58.163,-42.050,179.482,5.704,149.164
C08621=1183.731,-57.913,-42.061,179.485,5.704,149.164
C08622=1183.726,-57.663,-42.073,179.488,5.705,149.163
C08623=1183.720,-57.414,-42.084,179.489,5.705,149.163
C08624=1183.716,-57.164,-42.096,179.492,5.705,149.162
C08625=1183.711,-56.915,-42.107,179.495,5.706,149.161
C08626=1183.706,-56.665,-42.119,179.497,5.707,149.161
C08627=1183.700,-56.415,-42.129,179.499,5.706,149.160
C08628=1183.695,-56.165,-42.141,179.501,5.707,149.159
C08629=1183.690,-55.916,-42.152,179.504,5.707,149.159
C08630=1183.684,-55.666,-42.164,179.506,5.707,149.158
C08631=1183.680,-55.416,-42.175,179.508,5.708,149.157
C08632=1183.674,-55.167,-42.187,179.511,5.708,149.157
C08633=1183.669,-54.917,-42.198,179.513,5.709,149.156
C08634=1183.664,-54.668,-42.209,179.515,5.708,149.156
C08635=1183.659,-54.418,-42.221,179.518,5.709,149.155
C08636=1183.654,-54.168,-42.232,179.520,5.710,149.154
C08637=1183.648,-53.918,-42.243,179.522,5.709,149.154
C08638=1183.643,-53.669,-42.255,179.525,5.710,149.153
C08639=1183.638,-53.419,-42.267,179.527,5.711,149.152
C08640=1183.633,-53.169,-42.278,179.530,5.711,149.152
C08641=1183.628,-52.919,-42.290,179.532,5.711,149.151
C08642=1183.622,-52.670,-42.301,179.534,5.711,149.151
C08643=1183.617,-52.420,-42.313,179.537,5.712,149.150
C08644=1183.612,-52.170,-42.324,179.539,5.712,149.149
C08645=1183.607,-51.921,-42.336,179.541,5.712,149.148
C08646=1183.601,-51.671,-42.348,179.544,5.713,149.148
C08647=1183.597,-51.421,-42.359,179.546,5.713,149.147
C08648=1183.591,-51.172,-42.370,179.548,5.713,149.147
C08649=1183.586,-50.922,-42.382,179.551,5.714,149.146
C08650=1183.581,-50.672,-42.394,179.553,5.714,149.145
C08651=1183.575,-50.422,-42.405,179.556,5.714,149.145
C08652=1183.570,-50.173,-42.417,179.557,5.714,149.144
C08653=1183.565,-49.903,-42.429,179.560,5.715,149.144
C08654=1183.559,-49.633,-42.442,179.563,5.715,149.143
C08655=1183.554,-49.362,-42.455,179.566,5.716,149.142
C08656=1183.548,-49.092,-42.467,179.568,5.716,149.141
C08657=1183.542,-48.842,-42.479,179.571,5.717,149.141
C08658=1183.538,-48.593,-42.490,179.572,5.717,149.140
C08659=1183.532,-48.343,-42.502,179.575,5.717,149.140
C08660=1183.527,-48.093,-42.514,179.578,5.717,149.139
C08661=1183.522,-47.844,-42.526,179.580,5.718,149.138
C08662=1183.517,-47.594,-42.538,179.582,5.718,149.138
C08663=1183.511,-47.345,-42.550,179.585,5.718,149.137
C08664=1183.506,-47.095,-42.561,179.587,5.719,149.136
C08665=1183.501,-46.845,-42.573,179.590,5.720,149.136
C08666=1183.496,-46.595,-42.584,179.592,5.719,149.135
C08667=1183.491,-46.345,-42.596,179.594,5.720,149.134
C08668=1183.485,-46.096,-42.608,179.596,5.720,149.134
C08669=1183.481,-45.847,-42.620,179.599,5.721,149.133
C08670=1183.475,-45.597,-42.632,179.601,5.721,149.132
C08671=1183.470,-45.347,-42.644,179.604,5.721,149.132
C08672=1183.465,-45.097,-42.655,179.606,5.722,149.131
C08673=1183.460,-44.847,-42.667,179.609,5.722,149.131
C08674=1183.454,-44.598,-42.679,179.611,5.722,149.130
C08675=1183.449,-44.349,-42.691,179.613,5.723,149.129
C08676=1183.444,-44.099,-42.702,179.616,5.723,149.129
C08677=1183.439,-43.849,-42.714,179.618,5.724,149.128
C08678=1183.433,-43.600,-42.727,179.620,5.724,149.128
C08679=1183.428,-43.350,-42.738,179.623,5.724,149.127
C08680=1183.423,-43.100,-42.750,179.625,5.724,149.126
C08681=1183.418,-42.850,-42.762,179.628,5.725,149.125
C08682=1183.413,-42.601,-42.774,179.630,5.726,149.125
C08683=1183.407,-42.351,-42.786,179.632,5.725,149.124
C08684=1183.403,-42.101,-42.797,179.635,5.726,149.124
C08685=1183.397,-41.852,-42.810,179.637,5.727,149.123
C08686=1183.392,-41.602,-42.822,179.640,5.727,149.122
C08687=1183.387,-41.352,-42.834,179.642,5.727,149.122
C08688=1183.382,-41.102,-42.845,179.644,5.727,149.121
C08689=1183.377,-40.853,-42.858,179.647,5.728,149.121
C08690=1183.371,-40.603,-42.870,179.649,5.728,149.120
C08691=1183.366,-40.353,-42.881,179.651,5.728,149.119
C08692=1183.362,-40.104,-42.893,179.653,5.729,149.119
C08693=1183.356,-39.854,-42.905,179.656,5.729,149.118
C08694=1183.351,-39.604,-42.917,179.659,5.730,149.117
C08695=1183.346,-39.355,-42.930,179.661,5.730,149.117
C08696=1183.340,-39.105,-42.942,179.663,5.730,149.116
C08697=1183.335,-38.856,-42.954,179.666,5.731,149.115
C08698=1183.330,-38.606,-42.966,179.668,5.731,149.115
C08699=1183.325,-38.356,-42.977,179.671,5.732,149.114
C08700=1183.320,-38.107,-42.990,179.673,5.732,149.113
C08701=1183.314,-37.857,-43.002,179.675,5.732,149.113
C08702=1183.309,-37.608,-43.015,179.677,5.733,149.112
C08703=1183.304,-37.358,-43.026,179.680,5.733,149.112
C08704=1183.298,-37.108,-43.038,179.683,5.734,149.111
C08705=1183.294,-36.859,-43.050,179.685,5.734,149.110
C08706=1183.289,-36.609,-43.062,179.687,5.734,149.110
C08707=1183.283,-36.360,-43.075,179.690,5.735,149.109
C08708=1183.278,-36.110,-43.087,179.692,5.735,149.108
C08709=1183.273,-35.860,-43.099,179.695,5.736,149.108
C08710=1183.267,-35.610,-43.111,179.697,5.736,149.107
C08711=1183.262,-35.361,-43.124,179.699,5.736,149.106
C08712=1183.258,-35.110,-43.136,179.702,5.736,149.106
C08713=1183.252,-34.861,-43.149,179.704,5.737,149.105
C08714=1183.247,-34.611,-43.161,179.707,5.738,149.105
C08715=1183.243,-34.362,-43.173,179.709,5.738,149.104
C08716=1183.237,-34.112,-43.184,179.711,5.738,149.103
C08717=1183.232,-33.863,-43.197,179.714,5.739,149.103
C08718=1183.227,-33.613,-43.209,179.716,5.739,149.102
C08719=1183.221,-33.364,-43.222,179.719,5.739,149.101
C08720=1183.216,-33.114,-43.233,179.721,5.740,149.101
C08721=1183.211,-32.864,-43.246,179.723,5.740,149.100
C08722=1183.206,-32.615,-43.259,179.726,5.740,149.099
C08723=1183.200,-32.365,-43.271,179.728,5.741,149.099
C08724=1183.196,-32.115,-43.283,179.731,5.742,149.098
C08725=1183.190,-31.865,-43.295,179.733,5.742,149.098
C08726=1183.185,-31.616,-43.308,179.736,5.742,149.097
C08727=1183.180,-31.367,-43.321,179.738,5.743,149.096
C08728=1183.175,-31.117,-43.332,179.740,5.743,149.096
C08729=1183.170,-30.867,-43.345,179.743,5.743,149.095
C08730=1183.164,-30.618,-43.358,179.745,5.744,149.095
C08731=1183.159,-30.368,-43.370,179.748,5.745,149.094
C08732=1183.155,-30.118,-43.382,179.750,5.744,149.093
C08733=1183.149,-29.868,-43.394,179.753,5.745,149.092
C08734=1183.144,-29.619,-43.407,179.755,5.746,149.092
C08735=1183.139,-29.369,-43.420,179.757,5.746,149.091
C08736=1183.133,-29.120,-43.431,179.760,5.747,149.091
C08737=1183.128,-28.870,-43.444,179.762,5.747,149.090
C08738=1183.124,-28.620,-43.457,179.764,5.747,149.089
C08739=1183.119,-28.371,-43.470,179.767,5.747,149.089
C08740=1183.113,-28.121,-43.482,179.770,5.748,149.088
C08741=1183.108,-27.872,-43.494,179.772,5.749,149.088
C08742=1183.103,-27.622,-43.507,179.775,5.749,149.087
C08743=1183.097,-27.372,-43.519,179.777,5.750,149.086
C08744=1183.092,-27.122,-43.532,179.779,5.750,149.086
C08745=1183.087,-26.873,-43.545,179.781,5.750,149.085
C08746=1183.082,-26.623,-43.557,179.784,5.751,149.084
C08747=1183.077,-26.374,-43.570,179.787,5.751,149.084
C08748=1183.071,-26.124,-43.582,179.789,5.752,149.083
C08749=1183.067,-25.874,-43.595,179.792,5.752,149.082
C08750=1183.062,-25.625,-43.607,179.794,5.752,149.082
C08751=1183.057,-25.375,-43.620,179.796,5.753,149.081
C08752=1183.051,-25.126,-43.632,179.799,5.753,149.081
C08753=1183.046,-24.875,-43.645,179.801,5.754,149.080
C08754=1183.041,-24.626,-43.658,179.804,5.754,149.079
C08755=1183.036,-24.377,-43.671,179.806,5.755,149.079
C08756=1183.031,-24.127,-43.683,179.809,5.755,149.078
C08757=1183.026,-23.858,-43.697,179.811,5.756,149.077
C08758=1183.020,-23.587,-43.711,179.814,5.756,149.077
C08759=1183.014,-23.318,-43.724,179.817,5.757,149.076
C08760=1183.008,-23.048,-43.738,179.819,5.757,149.075
C08761=1183.003,-22.798,-43.751,179.821,5.757,149.075
C08762=1182.998,-22.549,-43.763,179.824,5.758,149.074
C08763=1182.993,-22.299,-43.776,179.826,5.758,149.073
C08764=1182.988,-22.050,-43.789,179.829,5.759,149.073
C08765=1182.983,-21.800,-43.802,179.831,5.759,149.072
C08766=1182.977,-21.551,-43.815,179.834,5.760,149.072
C08767=1182.973,-21.301,-43.828,179.836,5.760,149.071
C08768=1182.967,-21.051,-43.840,179.838,5.760,149.070
C08769=1182.962,-20.802,-43.852,179.841,5.761,149.070
C08770=1182.956,-20.552,-43.865,179.843,5.761,149.069
C08771=1182.952,-20.302,-43.878,179.846,5.762,149.068
C08772=1182.947,-20.053,-43.891,179.848,5.763,149.068
C08773=1182.942,-19.803,-43.903,179.851,5.763,149.067
C08774=1182.936,-19.553,-43.917,179.853,5.764,149.066
C08775=1182.931,-19.304,-43.930,179.856,5.764,149.066
C08776=1182.926,-19.054,-43.942,179.858,5.764,149.065
C08777=1182.922,-18.804,-43.955,179.860,5.764,149.065
C08778=1182.916,-18.555,-43.968,179.863,5.765,149.064
C08779=1182.911,-18.305,-43.981,179.865,5.766,149.063
C08780=1182.906,-18.056,-43.994,179.868,5.766,149.063
C08781=1182.900,-17.806,-44.007,179.871,5.767,149.062
C08782=1182.895,-17.556,-44.020,179.873,5.768,149.062
C08783=1182.890,-17.307,-44.032,179.875,5.768,149.061
C08784=1182.885,-17.057,-44.046,179.877,5.768,149.060
C08785=1182.880,-16.808,-44.059,179.880,5.768,149.059
C08786=1182.875,-16.559,-44.072,179.882,5.769,149.059
C08787=1182.870,-16.309,-44.085,179.885,5.769,149.058
C08788=1182.864,-16.059,-44.098,179.888,5.770,149.058
C08789=1182.860,-15.809,-44.111,179.890,5.771,149.057
C08790=1182.855,-15.560,-44.124,179.892,5.771,149.056
C08791=1182.849,-15.310,-44.137,179.895,5.772,149.056
C08792=1182.844,-15.060,-44.150,179.898,5.772,149.055
C08793=1182.839,-14.811,-44.163,179.899,5.772,149.055
C08794=1182.833,-14.561,-44.176,179.902,5.773,149.054
C08795=1182.829,-14.312,-44.189,179.905,5.773,149.053
C08796=1182.823,-14.062,-44.202,179.907,5.774,149.053
C08797=1182.819,-13.812,-44.215,179.909,5.774,149.052
C08798=1182.814,-13.563,-44.228,179.912,5.775,149.051
C08799=1182.808,-13.313,-44.241,179.915,5.775,149.051
C08800=1182.803,-13.063,-44.254,179.917,5.776,149.050
C08801=1182.798,-12.814,-44.268,179.920,5.777,149.050
C08802=1182.793,-12.565,-44.281,179.922,5.777,149.049
C08803=1182.788,-12.315,-44.294,179.924,5.778,149.048
C08804=1182.782,-12.065,-44.307,179.926,5.777,149.048
C08805=1182.778,-11.816,-44.321,179.929,5.778,149.047
C08806=1182.772,-11.566,-44.334,179.932,5.778,149.046
C08807=1182.768,-11.316,-44.347,179.934,5.779,149.046
C08808=1182.762,-11.067,-44.360,179.937,5.780,149.045
C08809=1182.757,-10.818,-44.373,179.939,5.780,149.044
C08810=1182.752,-10.568,-44.386,179.941,5.781,149.044
C08811=1182.747,-10.318,-44.399,179.944,5.781,149.043
C08812=1182.742,-10.068,-44.412,179.947,5.782,149.043
C08813=1182.737,-9.819,-44.426,179.949,5.782,149.042
C08814=1182.732,-9.569,-44.439,179.952,5.783,149.041
C08815=1182.726,-9.320,-44.452,179.954,5.784,149.041
C08816=1182.722,-9.070,-44.466,179.956,5.783,149.040
C08817=1182.716,-8.820,-44.479,179.958,5.784,149.040
C08818=1182.712,-8.570,-44.492,179.961,5.785,149.039
C08819=1182.706,-8.321,-44.506,179.964,5.785,149.038
C08820=1182.701,-8.072,-44.519,179.966,5.786,149.038
C08821=1182.696,-7.822,-44.532,179.969,5.786,149.037
C08822=1182.691,-7.573,-44.546,179.971,5.787,149.036
C08823=1182.685,-7.323,-44.559,179.974,5.787,149.036
C08824=1182.680,-7.073,-44.572,179.976,5.788,149.035
C08825=1182.675,-6.824,-44.586,179.979,5.789,149.035
C08826=1182.670,-6.574,-44.599,179.981,5.789,149.034
C08827=1182.665,-6.325,-44.613,179.984,5.790,149.033
C08828=1182.660,-6.075,-44.626,179.986,5.790,149.033
C08829=1182.655,-5.825,-44.639,179.989,5.791,149.032
C08830=1182.649,-5.576,-44.653,179.992,5.791,149.031
C08831=1182.645,-5.326,-44.666,179.993,5.791,149.031
C08832=1182.639,-5.077,-44.680,179.996,5.792,149.030
C08833=1182.635,-4.827,-44.693,179.998,5.792,149.029
C08834=1182.629,-4.578,-44.707,-179.999,5.793,149.029
C08835=1182.624,-4.328,-44.720,-179.997,5.794,149.028
C08836=1182.620,-4.078,-44.734,-179.994,5.794,149.028
C08837=1182.614,-3.829,-44.747,-179.991,5.795,149.027
C08838=1182.610,-3.579,-44.761,-179.989,5.795,149.026
C08839=1182.604,-3.330,-44.774,-179.987,5.796,149.026
C08840=1182.599,-3.080,-44.788,-179.984,5.796,149.025
C08841=1182.594,-2.831,-44.801,-179.981,5.797,149.024
C08842=1182.589,-2.581,-44.815,-179.979,5.798,149.024
C08843=1182.583,-2.331,-44.828,-179.976,5.798,149.023
C08844=1182.579,-2.082,-44.842,-179.974,5.799,149.023
C08845=1182.573,-1.832,-44.856,-179.972,5.799,149.022
C08846=1182.569,-1.583,-44.869,-179.969,5.800,149.021
C08847=1182.563,-1.332,-44.883,-179.966,5.800,149.021
C08848=1182.558,-1.083,-44.896,-179.964,5.801,149.020
C08849=1182.553,-0.834,-44.911,-179.961,5.802,149.020
C08850=1182.548,-0.584,-44.923,-179.959,5.802,149.019
C08851=1182.543,-0.335,-44.938,-179.956,5.803,149.018
C08852=1182.538,-0.084,-44.951,-179.954,5.804,149.018
C08853=1182.533,0.164,-44.965,-179.951,5.804,149.017
C08854=1182.528,0.414,-44.979,-179.949,5.804,149.016
C08855=1182.522,0.664,-44.992,-179.947,5.805,149.016
C08856=1182.518,0.913,-45.006,-179.944,5.805,149.015
C08857=1182.512,1.163,-45.019,-179.942,5.805,149.014
C08858=1182.507,1.412,-45.033,-179.939,5.806,149.014
C08859=1182.502,1.662,-45.047,-179.937,5.807,149.013
C08860=1182.497,1.911,-45.060,-179.934,5.807,149.013
C08861=1182.491,2.181,-45.075,-179.931,5.809,149.012
C08862=1182.486,2.450,-45.090,-179.928,5.809,149.011
C08863=1182.480,2.720,-45.105,-179.926,5.809,149.011
C08864=1182.475,2.988,-45.121,-179.923,5.810,149.010
C08865=1182.469,3.238,-45.134,-179.921,5.811,149.009
C08866=1182.465,3.488,-45.148,-179.918,5.811,149.009
C08867=1182.460,3.737,-45.162,-179.916,5.812,149.008
C08868=1182.454,3.987,-45.175,-179.913,5.813,149.008
C08869=1182.450,4.237,-45.189,-179.911,5.813,149.007
C08870=1182.444,4.486,-45.203,-179.908,5.814,149.006
C08871=1182.440,4.735,-45.217,-179.906,5.814,149.006
C08872=1182.434,4.985,-45.230,-179.903,5.815,149.005
C08873=1182.430,5.235,-45.245,-179.901,5.815,149.004
C08874=1182.424,5.484,-45.259,-179.898,5.816,149.004
C08875=1182.419,5.734,-45.273,-179.896,5.817,149.003
C08876=1182.414,5.983,-45.287,-179.893,5.817,149.003
C08877=1182.409,6.233,-45.300,-179.891,5.818,149.002
C08878=1182.404,6.482,-45.314,-179.888,5.818,149.001
C08879=1182.399,6.732,-45.328,-179.886,5.819,149.001
C08880=1182.393,6.981,-45.342,-179.883,5.819,149.000
C08881=1182.389,7.231,-45.357,-179.881,5.820,149.000
C08882=1182.384,7.481,-45.371,-179.878,5.821,148.999
C08883=1182.379,7.730,-45.385,-179.876,5.821,148.998
C08884=1182.373,7.980,-45.398,-179.873,5.822,148.998
C08885=1182.369,8.229,-45.412,-179.871,5.823,148.997
C08886=1182.364,8.479,-45.426,-179.868,5.823,148.996
C08887=1182.358,8.728,-45.440,-179.866,5.824,148.996
C08888=1182.353,8.978,-45.454,-179.863,5.824,148.995
C08889=1182.348,9.227,-45.469,-179.861,5.825,148.995
C08890=1182.343,9.477,-45.483,-179.858,5.825,148.994
C08891=1182.338,9.726,-45.497,-179.856,5.826,148.993
C08892=1182.333,9.976,-45.511,-179.853,5.827,148.993
C08893=1182.328,10.226,-45.525,-179.851,5.827,148.992
C08894=1182.323,10.475,-45.540,-179.848,5.828,148.992
C08895=1182.317,10.724,-45.554,-179.846,5.828,148.991
C08896=1182.312,10.974,-45.568,-179.843,5.829,148.990
C08897=1182.308,11.223,-45.582,-179.840,5.829,148.990
C08898=1182.303,11.473,-45.596,-179.838,5.830,148.989
C08899=1182.297,11.722,-45.610,-179.836,5.831,148.988
C08900=1182.293,11.972,-45.624,-179.833,5.831,148.988
C08901=1182.288,12.222,-45.638,-179.831,5.832,148.987
C08902=1182.283,12.471,-45.653,-179.828,5.833,148.987
C08903=1182.278,12.721,-45.667,-179.826,5.833,148.986
C08904=1182.272,12.970,-45.681,-179.823,5.834,148.985
C08905=1182.267,13.220,-45.695,-179.821,5.834,148.985
C08906=1182.262,13.469,-45.709,-179.817,5.836,148.984
C08907=1182.257,13.719,-45.724,-179.815,5.837,148.984
C08908=1182.252,13.969,-45.738,-179.813,5.837,148.983
C08909=1182.247,14.218,-45.752,-179.810,5.838,148.982
C08910=1182.241,14.468,-45.767,-179.807,5.838,148.982
C08911=1182.236,14.718,-45.781,-179.805,5.839,148.981
C08912=1182.231,14.967,-45.795,-179.803,5.839,148.980
C08913=1182.226,15.217,-45.810,-179.800,5.840,148.980
C08914=1182.222,15.466,-45.825,-179.798,5.841,148.979
C08915=1182.216,15.715,-45.838,-179.795,5.841,148.979
C08916=1182.211,15.965,-45.853,-179.792,5.842,148.978
C08917=1182.206,16.214,-45.867,-179.790,5.843,148.977
C08918=1182.201,16.464,-45.881,-179.788,5.843,148.977
C08919=1182.196,16.714,-45.896,-179.785,5.844,148.976
C08920=1182.191,16.964,-45.910,-179.783,5.844,148.976
C08921=1182.187,17.213,-45.925,-179.780,5.845,148.975
C08922=1182.181,17.462,-45.939,-179.777,5.845,148.974
C08923=1182.175,17.712,-45.954,-179.775,5.846,148.974
C08924=1182.170,17.961,-45.968,-179.772,5.847,148.973
C08925=1182.165,18.211,-45.982,-179.769,5.848,148.972
C08926=1182.161,18.460,-45.997,-179.767,5.849,148.972
C08927=1182.156,18.710,-46.011,-179.765,5.849,148.971
C08928=1182.151,18.960,-46.026,-179.762,5.850,148.971
C08929=1182.146,19.209,-46.040,-179.760,5.851,148.970
C08930=1182.141,19.458,-46.055,-179.757,5.851,148.969
C08931=1182.135,19.708,-46.070,-179.755,5.852,148.969
C08932=1182.130,19.958,-46.084,-179.752,5.852,148.968
C08933=1182.125,20.207,-46.099,-179.750,5.853,148.968
C08934=1182.120,20.456,-46.113,-179.747,5.853,148.967
C08935=1182.115,20.706,-46.127,-179.744,5.854,148.966
C08936=1182.110,20.956,-46.142,-179.742,5.855,148.966
C08937=1182.105,21.205,-46.157,-179.740,5.855,148.965
C08938=1182.100,21.455,-46.171,-179.736,5.857,148.965
C08939=1182.095,21.705,-46.186,-179.734,5.857,148.964
C08940=1182.091,21.954,-46.201,-179.732,5.858,148.963
C08941=1182.085,22.204,-46.216,-179.729,5.858,148.963
C08942=1182.080,22.453,-46.230,-179.727,5.859,148.962
C08943=1182.075,22.702,-46.245,-179.724,5.860,148.962
C08944=1182.070,22.952,-46.259,-179.721,5.860,148.961
C08945=1182.064,23.201,-46.274,-179.719,5.861,148.960
C08946=1182.059,23.451,-46.289,-179.717,5.862,148.960
C08947=1182.054,23.700,-46.303,-179.714,5.862,148.959
C08948=1182.050,23.949,-46.318,-179.712,5.863,148.959
C08949=1182.044,24.199,-46.333,-179.709,5.864,148.958
C08950=1182.039,24.449,-46.348,-179.706,5.865,148.957
C08951=1182.034,24.698,-46.362,-179.704,5.866,148.957
C08952=1182.030,24.947,-46.377,-179.701,5.866,148.956
C08953=1182.024,25.197,-46.392,-179.699,5.867,148.955
C08954=1182.019,25.446,-46.407,-179.696,5.867,148.955
C08955=1182.014,25.696,-46.421,-179.694,5.868,148.954
C08956=1182.009,25.946,-46.436,-179.691,5.868,148.954
C08957=1182.004,26.195,-46.451,-179.689,5.869,148.953
C08958=1181.999,26.445,-46.465,-179.686,5.871,148.953
C08959=1181.994,26.694,-46.481,-179.683,5.871,148.952
C08960=1181.989,26.944,-46.495,-179.681,5.872,148.951
C08961=1181.984,27.193,-46.510,-179.678,5.872,148.951
C08962=1181.979,27.443,-46.526,-179.676,5.873,148.950
C08963=1181.974,27.692,-46.540,-179.673,5.874,148.950
C08964=1181.969,27.941,-46.555,-179.671,5.874,148.949
C08965=1181.963,28.210,-46.571,-179.668,5.876,148.948
C08966=1181.958,28.479,-46.587,-179.665,5.876,148.948
C08967=1181.952,28.748,-46.603,-179.663,5.877,148.947
C08968=1181.947,29.017,-46.619,-179.660,5.878,148.946
C08969=1181.942,29.267,-46.635,-179.657,5.879,148.946
C08970=1181.937,29.516,-46.649,-179.654,5.879,148.945
C08971=1181.933,29.766,-46.664,-179.652,5.880,148.945
C08972=1181.927,30.015,-46.680,-179.649,5.881,148.944
C08973=1181.922,30.265,-46.694,-179.647,5.881,148.943
C08974=1181.917,30.515,-46.710,-179.645,5.882,148.943
C08975=1181.912,30.764,-46.725,-179.642,5.883,148.942
C08976=1181.907,31.013,-46.739,-179.639,5.883,148.941
C08977=1181.902,31.263,-46.755,-179.637,5.885,148.941
C08978=1181.897,31.512,-46.770,-179.634,5.885,148.940
C08979=1181.892,31.762,-46.784,-179.631,5.886,148.940
C08980=1181.887,32.011,-46.799,-179.629,5.887,148.939
C08981=1181.882,32.260,-46.815,-179.626,5.887,148.939
C08982=1181.877,32.511,-46.830,-179.624,5.888,148.938
C08983=1181.872,32.760,-46.845,-179.622,5.888,148.937
C08984=1181.867,33.009,-46.860,-179.618,5.890,148.937
C08985=1181.862,33.259,-46.876,-179.616,5.891,148.936
C08986=1181.857,33.508,-46.890,-179.614,5.891,148.936
C08987=1181.852,33.758,-46.906,-179.611,5.892,148.935
C08988=1181.847,34.007,-46.921,-179.609,5.892,148.934
C08989=1181.842,34.256,-46.936,-179.606,5.893,148.934
C08990=1181.837,34.507,-46.951,-179.603,5.894,148.933
C08991=1181.832,34.756,-46.967,-179.601,5.895,148.933
C08992=1181.827,35.005,-46.982,-179.598,5.896,148.932
C08993=1181.822,35.255,-46.997,-179.596,5.896,148.931
C08994=1181.817,35.504,-47.012,-179.593,5.897,148.931
C08995=1181.812,35.753,-47.028,-179.591,5.898,148.930
C08996=1181.807,36.003,-47.042,-179.589,5.898,148.930
C08997=1181.802,36.253,-47.058,-179.585,5.900,148.929
C08998=1181.797,36.502,-47.074,-179.583,5.900,148.928
C08999=1181.792,36.751,-47.089,-179.581,5.901,148.928
C09000=1181.787,37.001,-47.104,-179.578,5.902,148.927
C09001=1181.782,37.250,-47.119,-179.575,5.902,148.927
C09002=1181.777,37.500,-47.135,-179.573,5.904,148.926
C09003=1181.771,37.750,-47.150,-179.570,5.904,148.925
C09004=1181.767,37.999,-47.165,-179.567,5.905,148.925
C09005=1181.761,38.249,-47.181,-179.565,5.906,148.924
C09006=1181.757,38.498,-47.196,-179.562,5.906,148.924
C09007=1181.751,38.747,-47.211,-179.560,5.907,148.923
C09008=1181.747,38.997,-47.227,-179.557,5.908,148.923
C09009=1181.742,39.246,-47.242,-179.554,5.909,148.922
C09010=1181.737,39.496,-47.258,-179.552,5.910,148.921
C09011=1181.731,39.745,-47.273,-179.550,5.910,148.921
C09012=1181.727,39.995,-47.289,-179.547,5.911,148.920
C09013=1181.722,40.244,-47.304,-179.544,5.912,148.920
C09014=1181.716,40.494,-47.320,-179.542,5.913,148.919
C09015=1181.712,40.743,-47.335,-179.539,5.913,148.918
C09016=1181.707,40.993,-47.351,-179.537,5.914,148.918
C09017=1181.702,41.242,-47.366,-179.534,5.915,148.917
C09018=1181.697,41.491,-47.381,-179.531,5.916,148.917
C09019=1181.692,41.741,-47.397,-179.529,5.917,148.916
C09020=1181.687,41.991,-47.413,-179.526,5.917,148.915
C09021=1181.681,42.240,-47.428,-179.524,5.918,148.915
C09022=1181.677,42.489,-47.443,-179.521,5.919,148.914
C09023=1181.671,42.739,-47.459,-179.518,5.920,148.914
C09024=1181.667,42.989,-47.475,-179.516,5.921,148.913
C09025=1181.662,43.238,-47.490,-179.513,5.922,148.913
C09026=1181.656,43.487,-47.506,-179.511,5.922,148.912
C09027=1181.651,43.736,-47.522,-179.509,5.923,148.911
C09028=1181.647,43.986,-47.538,-179.505,5.924,148.911
C09029=1181.642,44.235,-47.553,-179.503,5.925,148.910
C09030=1181.637,44.485,-47.568,-179.500,5.926,148.910
C09031=1181.632,44.735,-47.584,-179.498,5.926,148.909
C09032=1181.626,44.984,-47.600,-179.496,5.927,148.908
C09033=1181.621,45.234,-47.615,-179.492,5.928,148.908
C09034=1181.617,45.483,-47.632,-179.490,5.929,148.907
C09035=1181.612,45.732,-47.647,-179.488,5.930,148.907
C09036=1181.607,45.982,-47.663,-179.485,5.930,148.906
C09037=1181.602,46.232,-47.679,-179.482,5.932,148.906
C09038=1181.596,46.481,-47.694,-179.480,5.932,148.905
C09039=1181.592,46.730,-47.710,-179.478,5.933,148.904
C09040=1181.587,46.980,-47.726,-179.475,5.934,148.904
C09041=1181.582,47.229,-47.742,-179.472,5.934,148.903
C09042=1181.576,47.478,-47.757,-179.469,5.936,148.903
C09043=1181.572,47.729,-47.773,-179.467,5.937,148.902
C09044=1181.567,47.977,-47.789,-179.465,5.937,148.902
C09045=1181.562,48.226,-47.804,-179.462,5.938,148.901
C09046=1181.557,48.477,-47.820,-179.459,5.939,148.900
C09047=1181.552,48.725,-47.837,-179.457,5.940,148.900
C09048=1181.547,48.975,-47.853,-179.454,5.941,148.899
C09049=1181.542,49.225,-47.868,-179.452,5.941,148.899
C09050=1181.537,49.474,-47.884,-179.449,5.943,148.898
C09051=1181.532,49.724,-47.900,-179.446,5.943,148.897
C09052=1181.527,49.973,-47.916,-179.444,5.944,148.897
C09053=1181.522,50.223,-47.933,-179.441,5.945,148.896
C09054=1181.517,50.472,-47.948,-179.439,5.946,148.896
C09055=1181.512,50.721,-47.963,-179.436,5.947,148.895
C09056=1181.508,50.971,-47.980,-179.433,5.947,148.894
C09057=1181.502,51.220,-47.996,-179.431,5.948,148.894
C09058=1181.497,51.470,-48.011,-179.428,5.950,148.893
C09059=1181.492,51.719,-48.028,-179.426,5.951,148.893
C09060=1181.487,51.968,-48.043,-179.423,5.951,148.892
C09061=1181.483,52.218,-48.060,-179.420,5.952,148.892
C09062=1181.477,52.467,-48.076,-179.418,5.953,148.891
C09063=1181.472,52.717,-48.092,-179.415,5.954,148.890
C09064=1181.467,52.966,-48.108,-179.413,5.955,148.890
C09065=1181.462,53.216,-48.124,-179.410,5.955,148.889
C09066=1181.457,53.465,-48.140,-179.407,5.956,148.889
C09067=1181.453,53.715,-48.156,-179.405,5.957,148.888
C09068=1181.448,53.964,-48.172,-179.402,5.958,148.888
C09069=1181.442,54.232,-48.189,-179.399,5.959,148.887
C09070=1181.437,54.501,-48.207,-179.397,5.960,148.886
C09071=1181.432,54.769,-48.225,-179.394,5.961,148.886
C09072=1181.426,55.038,-48.242,-179.391,5.962,148.885
C09073=1181.421,55.288,-48.257,-179.389,5.963,148.885
C09074=1181.416,55.537,-48.274,-179.386,5.964,148.884
C09075=1181.412,55.787,-48.290,-179.383,5.965,148.883
C09076=1181.406,56.036,-48.307,-179.381,5.966,148.883
C09077=1181.401,56.285,-48.323,-179.378,5.966,148.882
C09078=1181.396,56.535,-48.339,-179.376,5.968,148.882
C09079=1181.391,56.784,-48.356,-179.373,5.968,148.881
C09080=1181.386,57.034,-48.371,-179.370,5.969,148.881
C09081=1181.382,57.283,-48.388,-179.368,5.970,148.880
C09082=1181.376,57.532,-48.404,-179.365,5.971,148.879
C09083=1181.372,57.782,-48.420,-179.363,5.972,148.879
C09084=1181.367,58.031,-48.436,-179.360,5.972,148.878
C09085=1181.362,58.281,-48.452,-179.357,5.974,148.878
C09086=1181.357,58.530,-48.469,-179.355,5.975,148.877
C09087=1181.351,58.780,-48.486,-179.352,5.975,148.877
C09088=1181.346,59.029,-48.501,-179.349,5.977,148.876
C09089=1181.342,59.278,-48.518,-179.347,5.977,148.875
C09090=1181.337,59.527,-48.534,-179.345,5.978,148.875
C09091=1181.332,59.777,-48.550,-179.341,5.980,148.874
C09092=1181.327,60.027,-48.567,-179.339,5.980,148.874
C09093=1181.321,60.276,-48.584,-179.337,5.981,148.873
C09094=1181.317,60.525,-48.601,-179.334,5.982,148.873
C09095=1181.312,60.775,-48.616,-179.331,5.983,148.872
C09096=1181.307,61.024,-48.633,-179.329,5.984,148.871
C09097=1181.302,61.273,-48.649,-179.326,5.985,148.871
C09098=1181.297,61.523,-48.665,-179.323,5.986,148.870
C09099=1181.292,61.773,-48.682,-179.321,5.987,148.870
C09100=1181.287,62.022,-48.699,-179.318,5.987,148.869
C09101=1181.282,62.271,-48.715,-179.316,5.989,148.869
C09102=1181.277,62.520,-48.732,-179.313,5.990,148.868
C09103=1181.272,62.770,-48.748,-179.310,5.990,148.868
C09104=1181.267,63.020,-48.765,-179.308,5.992,148.867
C09105=1181.262,63.269,-48.781,-179.305,5.992,148.866
C09106=1181.258,63.518,-48.798,-179.303,5.993,148.866
C09107=1181.253,63.768,-48.815,-179.300,5.995,148.865
C09108=1181.248,64.017,-48.831,-179.298,5.995,148.865
C09109=1181.243,64.267,-48.847,-179.295,5.996,148.864
C09110=1181.238,64.516,-48.864,-179.292,5.998,148.864
C09111=1181.232,64.765,-48.881,-179.290,5.998,148.863
C09112=1181.228,65.015,-48.898,-179.287,5.999,148.863
C09113=1181.223,65.264,-48.914,-179.284,6.000,148.862
C09114=1181.218,65.513,-48.931,-179.282,6.001,148.861
C09115=1181.213,65.763,-48.948,-179.279,6.002,148.861
C09116=1181.208,66.012,-48.964,-179.276,6.003,148.860
C09117=1181.204,66.261,-48.981,-179.274,6.004,148.860
C09118=1181.198,66.511,-48.998,-179.271,6.005,148.859
C09119=1181.193,66.760,-49.014,-179.269,6.006,148.859
C09120=1181.189,67.010,-49.030,-179.266,6.007,148.858
C09121=1181.183,67.260,-49.048,-179.264,6.008,148.858
C09122=1181.178,67.508,-49.064,-179.261,6.009,148.857
C09123=1181.173,67.758,-49.081,-179.259,6.010,148.857
C09124=1181.169,68.008,-49.098,-179.256,6.010,148.856
C09125=1181.164,68.257,-49.115,-179.253,6.012,148.855
C09126=1181.158,68.506,-49.131,-179.251,6.013,148.855
C09127=1181.154,68.756,-49.148,-179.247,6.014,148.854
C09128=1181.149,69.005,-49.165,-179.245,6.015,148.854
C09129=1181.144,69.254,-49.182,-179.243,6.015,148.853
C09130=1181.139,69.503,-49.199,-179.240,6.017,148.853
C09131=1181.134,69.753,-49.216,-179.237,6.018,148.852
C09132=1181.130,70.003,-49.233,-179.235,6.019,148.852
C09133=1181.124,70.251,-49.249,-179.232,6.020,148.851
C09134=1181.119,70.501,-49.267,-179.230,6.021,148.850
C09135=1181.115,70.751,-49.283,-179.227,6.021,148.850
C09136=1181.110,71.000,-49.301,-179.224,6.023,148.849
C09137=1181.104,71.249,-49.317,-179.222,6.024,148.849
C09138=1181.099,71.499,-49.334,-179.219,6.025,148.848
C09139=1181.095,71.748,-49.351,-179.216,6.026,148.848
C09140=1181.090,71.998,-49.369,-179.214,6.027,148.847
C09141=1181.085,72.246,-49.385,-179.211,6.028,148.847
C09142=1181.080,72.496,-49.402,-179.209,6.029,148.846
C09143=1181.075,72.746,-49.419,-179.206,6.030,148.845
C09144=1181.070,72.995,-49.436,-179.203,6.031,148.845
C09145=1181.065,73.244,-49.453,-179.201,6.032,148.844
C09146=1181.060,73.493,-49.471,-179.198,6.033,148.844
C09147=1181.055,73.743,-49.487,-179.196,6.034,148.843
C09148=1181.050,73.993,-49.504,-179.193,6.034,148.843
C09149=1181.046,74.242,-49.521,-179.190,6.036,148.842
C09150=1181.040,74.491,-49.539,-179.188,6.037,148.842
